// TwinCAT 3 PLC project PLC_851
// Title: 2505
// Company: Infineon
// Author: Utz
// ProgramVersion: 3.1.4023.0
// CompilerDefines: VISU_USEPROPERTYINFO
// libraries:
//   GeneralLib, * (IB-Muhr)
//   CmpBitmapPool, * (System)
//   GeneralLib, * (IB-Muhr)
//   Tc2_EtherCAT, * (Beckhoff Automation GmbH)
//   Tc2_MC2, * (Beckhoff Automation GmbH)
//   Tc2_SerialCom, * (Beckhoff Automation GmbH)
//   Tc2_Standard, * (Beckhoff Automation GmbH)
//   Tc2_System, * (Beckhoff Automation GmbH)
//   Tc2_TcpIp, * (Beckhoff Automation GmbH)
//   Tc2_Utilities, * (Beckhoff Automation GmbH)
//   Tc2_XmlDataSrv, * (Beckhoff Automation GmbH)
//   Tc3_Database, * (Beckhoff Automation GmbH)
//   Tc3_EventLogger, * (Beckhoff Automation GmbH)
//   Tc3_IotBase, * (Beckhoff Automation GmbH)
//   Tc3_Module, * (Beckhoff Automation GmbH)
//   VisuDialogs, * (System)
//   VisuSymbols, * (System)
//   Tc2_Standard,3.3.3.0,Beckhoff Automation GmbH
//   VisuSymbols,3.5.10.0,System
// project tree:
//   DUTs/ ST_RECIPE_ENDURANCE_RUN.TcDUT, ST_RECIPE_BREAK_PRESSURE.TcDUT, ST_RECIPE_GENERAL.TcDUT, ST_RECIPE_LEAK_TEST1.TcDUT, ST_RECIPE_LEAK_TEST2.TcDUT, ST_RECIPE_PARAMS.TcDUT, ST_RECIPE_CYL.TcDUT, ST_SETTINGS.TcDUT
//   FUNCTIONS/FUNCTIONS/MATH/ F_RoundLREAL.TcPOU, F_RoundREAL.TcPOU
//   / GlobalTextList.TcGTLO, GVL.TcGVL, GVL_EventLogger.TcGVL, MeasureTask.TcTTO, PlcTask.TcTTO, ProjectInfo.TcGVL, TXT_LIST_OBJECTS.TcTLO, VisuTask.TcTTO
//   MODULE/ACTOR_VALVE/GENERAL/DUT/ E_POS_STATE.TcDUT, E_SPEED_TYPE.TcDUT, E_PRESSURE_TYPE.TcDUT, ST_CYL_CALIBRATION.TcDUT, ST_HMI_CYLINDER.TcDUT, ST_HMI_VALVE.TcDUT, ST_RECORD.TcDUT, ST_RECORD_DATA.TcDUT
//   MODULE/ACTOR_VALVE/HYDRAULIC_ACTOR/DUT/ E_SEQ_CYLINDER.TcDUT, E_SEQ_ENGINE.TcDUT
//   MODULE/ACTOR_VALVE/HYDRAULIC_ACTOR/ITF/ I_CYLINDER_DA_COUNTER.TcIO, I_CYLINDER_DA_GENERAL.TcIO, I_CYLINDER_DA_TESTDEV2_4.TcIO, I_CYLINDER_SA_GENERAL.TcIO, I_CYLINDER_DA_TESTDEV1.TcIO, I_ENGINE.TcIO, I_PUMP.TcIO, I_PUMP_WITH_BYPASS.TcIO
//   MODULE/ACTOR_VALVE/HYDRAULIC_ACTOR/POU/ FB_CYLINDER_DA_COUNTER.TcPOU, FB_CYLINDER_DA_TESTDEV1.TcPOU, FB_CYLINDER_DA_TESTDEV2_4.TcPOU, FB_PUMP.TcPOU, FB_PUMP_WITH_BYPASS.TcPOU
//   MODULE/ACTOR_VALVE/PNEUMATIC_ACTOR/DUT/ E_PNEU_VAC_VALVE.TcDUT
//   MODULE/ACTOR_VALVE/PNEUMATIC_ACTOR/ITF/ I_PNEU_ACTOR.TcIO, I_STOP_GATE.TcIO, I_VAC_VALVE.TcIO
//   MODULE/ACTOR_VALVE/PNEUMATIC_ACTOR/POU/ FB_STOP_GATE.TcPOU, FB_VAC_BLOW_VALVE.TcPOU, FB_VAC_VALVE.TcPOU, FB_VISU_CYLINDER.TcPOU, FB_VISU_STOP_GATE.TcPOU, FB_VISU_VAC_VALVE.TcPOU, FB_ZYLINDER_TWO_WAY.TcPOU, FB_ZYLINDER_TWO_WAY_MID_POS.TcPOU
//   MODULE/ACTOR_VALVE/PNEUMATIC_ACTOR/TXTLIST/ TXT_LIST_PNEMATIC_ACTOR.TcTLO
//   MODULE/ACTOR_VALVE/PNEUMATIC_ACTOR/VISU/ VisuCylinderGripperDown.TcVIS, VisuCylinderHorLeft.TcVIS, VisuCylinderHorLeftCtrl.TcVIS, VisuCylinderHorRight.TcVIS, VisuCylinderHorRightCtrl.TcVIS, VisuCylinderHorRight_MidPos.TcVIS, VisuCylinderTurn.TcVIS, VisuCylinderVertDown.TcVIS, VisuCylinderVertDownCtrl.TcVIS, VisuCylinderVertUp.TcVIS, VisuCylinderVertUpCtrl.TcVIS
//   MODULE/ACTOR_VALVE/VALVE/DUT/ E_SEQ_VALVE.TcDUT
//   MODULE/ACTOR_VALVE/VALVE/ITF/ I_ENGINE_VALVE.TcIO, I_PRV_PROP.TcIO, I_VALVE_X_3_PROP.TcIO, I_VALVE_X_2.TcIO, I_VALVE_X_3.TcIO
//   MODULE/ACTOR_VALVE/VALVE/POU/ FB_SHUTOFF_VALVE.TcPOU, FB_PRV_PROP.TcPOU, FB_VALVE_X_2.TcPOU, FB_VALVE_X_3.TcPOU, FB_VALVE_X_3_PROP.TcPOU
//   MODULE/BUS_DIAG/POU/ FB_EC_MASTER.TcPOU, FB_VISU_BUS_DIAG.TcPOU
//   MODULE/BUS_DIAG/VISU/ VISU_BUS_DIAG_MASTER.TcVIS
//   MODULE/BYTES_TO_WORD/DUT/ U_BytesToWord.TcDUT
//   MODULE/BYTES_TO_WORD/ITF/ I_WORD_TO_BYTES.TcIO
//   MODULE/BYTES_TO_WORD/POU/ FB_BYTES_TO_WORD.TcPOU, FB_WORD_TO_BYTES.TcPOU
//   MODULE/BYTES_TO_WORD/VISU/ FB_VISU_WORD_TO_BYTES.TcPOU, VISU_WORD_TO_BYTES.TcVIS
//   MODULE/DATABASE/DUT/ E_SEQ_DATABASE.TcDUT, ST_DATABASE_RECORD.TcDUT
//   MODULE/DATABASE/ITF/ I_DATABASE.TcIO, I_INFLUXDB_ADS.TcIO
//   MODULE/DATABASE/POU/ FB_INFLUX_DB.TcPOU, FB_INFLUX_DB_ADS.TcPOU, FB_MY_SQL.TcPOU
//   MODULE/FREQUENCE/ITF/ I_FREQ_GEN.TcIO
//   MODULE/FREQUENCE/POU/ FB_FREQENCE.TcPOU
//   MODULE/GENERAL/DUT/ E_STEP_STATE.TcDUT
//   MODULE/GENERAL/ E_Direction.TcDUT, F_Lineare_Regression.TcPOU, F_RangeSetpoint.TcPOU, stMesswerte.TcDUT, stRampAnalytic.TcDUT, ST_CHART.TcDUT
//   MODULE/GENERAL/INPUTS/ITF/ I_BINARY_SWITCH_SENS.TcIO
//   MODULE/GENERAL/INPUTS/POU/ FB_BINARY_SWITCH_SENS.TcPOU
//   MODULE/GENERAL/SIMU_ANALOG_IN/ FB_SIMU_ANALOG_IN.TcPOU, I_SIMU_ANALOG_IN.TcIO
//   MODULE/HMI/DUT/ E_SEQ_HMI.TcDUT
//   MODULE/HMI/ITF/ I_HMI_CTRL.TcIO
//   MODULE/HMI/POU/ FB_HMI_CTRL.TcPOU, FB_HMI_CTRL_ADS.TcPOU
//   MODULE/SAFETY/DUT/ E_STEP_STATE_ESTOP.TcDUT
//   MODULE/SAFETY/ GVL_SAFETY.TcGVL
//   MODULE/SAFETY/ITF/ I_ESTOP.TcIO
//   MODULE/SAFETY/PIC/ IMG_LIST_GATE_LOCK.TcIPO (not stored)
//   MODULE/SAFETY/POU/ FB_ESTOP.TcPOU
//   MODULE/SAFETY/VISU/ FB_VISU_GATE_LOCK.TcPOU
//   IMPLICIT_CHECKS/ CheckBounds.TcPOU, CheckDivDInt.TcPOU, CheckDivLInt.TcPOU, CheckDivLReal.TcPOU, CheckDivReal.TcPOU, CheckLRangeSigned.TcPOU, CheckLRangeUnsigned.TcPOU, CheckPointer.TcPOU, CheckRangeSigned.TcPOU, CheckRangeUnsigned.TcPOU
//   MODULE/TRAFFIC_LIGHT/ITFs/ I_TrafficLight.TcIO
//   MODULE/TRAFFIC_LIGHT/POUs/ FB_TrafficLight.TcPOU
//   ORGANISATION/DATE_TIME/ITF/ I_CLOCK.TcIO
//   ORGANISATION/DATE_TIME/POU/ FB_CLOCK.TcPOU
//   ORGANISATION/EVENT_LOGGER/ITFs/ I_EVENT_LOGGER.TcIO
//   ORGANISATION/EVENT_LOGGER/POUs/ FB_EVENT_LOGGER.TcPOU
//   ORGANISATION/GENERAL/DUT/ E_SEQ_GENERAL.TcTLEO, E_STEP_STATE_TYPE.TcDUT, ST_GENERAL_HMI.TcDUT, ST_LAST_STEPS.TcDUT, ST_SEQ_CTRL_GEN.TcDUT
//   ORGANISATION/GENERAL/ITF/ FB_Abstract_FunktionCtrl.TcPOU, I_FunctionCtrl.TcIO, I_GENERAL.TcIO
//   ORGANISATION/GENERAL/POU/ FB_GENERAL.TcPOU, F_CreateObjectName.TcPOU
//   ORGANISATION/OP_MODE/DUT/ ST_EVENT_DATA.TcDUT, ST_LOG_EVENT.TcDUT
//   ORGANISATION/OP_MODE/GVL_PARA/ OP_MODE.TcGVL
//   ORGANISATION/OP_MODE/ITF/ I_OP_MODE.TcIO, I_OP_MODE_PAUSE.TcIO, I_OP_MODE_PAUSE_VISU.TcIO
//   ORGANISATION/OP_MODE/POU/ FB_OP_MODE.TcPOU, FB_OP_MODE_HMI.TcPOU, FB_OP_MODE_PAUSE.TcPOU, FB_OP_MODE_PAUSE_VISU.TcPOU, FB_OP_MODE_VISU.TcPOU
//   ORGANISATION/OP_MODE/TXTLIST/ TXT_LIST_OP_MODE.TcTLO
//   ORGANISATION/USER_MANAGER/POU/ FB_ESTOP_RESET.TcPOU
//   POUs/ F_SEND_EVENTLOGGER_MSG.TcPOU, MAIN.TcPOU
//   PROGRAMS/ PrgMeasure.TcPOU, PrgOrg.TcPOU, PrgStation.TcPOU, PrgVisu.TcPOU
//   SUBSTATION/ GVL_SUBSTATION.TcGVL
//   SUBSTATION/STATION_NEST/DUT/ E_SEQ_PROCESS.TcDUT, ST_ENDURANCERUN_RECORD.TcDUT
//   SUBSTATION/STATION_NEST/ GVL_PROCESS.TcGVL
//   SUBSTATION/STATION_NEST/ITF/ I_PROCESS_MAIN.TcIO, I_PROCESS_NEST1.TcIO, I_PROCESS_NEST2_4.TcIO
//   SUBSTATION/STATION_NEST/POU/ FB_PROCESS_MAIN.TcPOU, FB_SEQ_PROCESS_NEST1.TcPOU, FB_SEQ_PROCESS_NEST2_4.TcPOU

CONFIGURATION PLC_851
    RESOURCE PLC ON TwinCAT3
        TASK MeasureTask(INTERVAL := T#10ms, PRIORITY := 2);
        TASK PlcTask(INTERVAL := T#10ms, PRIORITY := 21);
        TASK VisuTask(INTERVAL := T#100000us, PRIORITY := 1);
        PROGRAM PrgMeasure WITH MeasureTask : PrgMeasure;
        PROGRAM PrgStation WITH PlcTask : PrgStation;
        PROGRAM PrgOrg WITH PlcTask : PrgOrg;
        PROGRAM PrgVisu WITH VisuTask : PrgVisu;
    END_RESOURCE
END_CONFIGURATION

// ---- DUTs/ST_RECIPE_ENDURANCE_RUN.TcDUT
TYPE ST_RECIPE_ENDURANCE_RUN :
STRUCT
  // Enables
  bEnableVentCylinder:            BOOL;
  bEnableEnduranceRun:            BOOL;
  bEnableLeakTest1:               BOOL;
  // Vent cylinder
  uiVentCycles:                   UINT;
  // Profiles - Endurance run
  rSpeedA:                        REAL;         // Speed A
  rSpeedB:                        REAL;         // Speed B
  rWorkPressureA:                 REAL;         // Work pressure testing cylinder A
  rWorkPressureB:                 REAL;         // Work pressure testing cylinder B
  rWorkForceA:                    REAL;         // Work force testing cylinder A
  rWorkForceB:                    REAL;         // Work force testing cylinder B
  udiCycles:                      UDINT;        // Count of cycles
  rLoadPressureA:                 REAL;         // Load pressure A (counterload)
  rLoadPressureB:                 REAL;         // Load pressure B (counterload)
  rLoadForceA:                    REAL;         // Load force A (counterload)
  rLoadForceB:                    REAL;         // Load force B (counterload)
  rTurningPointHP:                REAL;         // Cylinder turning point in HP
  rTurningPointWP:                REAL;         // Cylinder turning point in WP
  rDelay:                         REAL;         // Delay on turning point
  // Quick leak test 1 parameter
  udiLT1_Interval:                UDINT;        // Interval for quick leak test 1
  stLT1_Params:                   ST_RECIPE_LEAK_TEST1;
  //rLT1_RestDelay:                 REAL;         // Rest delay aufter test
  //rLT1_LoadForceA:                REAL;         // Load force A (counterload)
  //rLT1_LoadForceB:                REAL;         // Load force B (counterload)
  //rLT1_LoadPressureA:             REAL;         // Testing pressure A for leak test 1
  //rLT1_LoadPressureB:             REAL;         // Testing pressure B for leak test 1
  //uiLT1_DurationPerTest:          UINT;         // Testing duration per test in min
  //rLT1_DistanceBeforeEndPosHP:    REAL;         // Distance to the end position HP
  //rLT1_DistanceBeforeEndPosWP:    REAL;         // Distance to the end position WP
  //rLT1_NokLimit:                  REAL;         // Delta length limit to abort program
END_STRUCT
END_TYPE

// ---- DUTs/ST_RECIPE_BREAK_PRESSURE.TcDUT
TYPE ST_RECIPE_BREAK_PRESSURE :
STRUCT
  // Enables
  bEnableVentCylinder:            BOOL;
  bEnableBreakPressureDet:        BOOL;
  // Vent cylinder
  uiVentCycles:                   UINT;
  // Break pressure determination
  rMinSpeedInMmPerS:              REAL;         // Minimal speed in mm/s
  rEndPosTol:                     REAL;         // End position tolerance
  rIncreaseInterval:              REAL;         // Interval in seconds
  rIncreaseValueInBar:            REAL;         // Value in bar to increase if not mooving
  rNokLimit:                      REAL;         // Pressure limit to abort
END_STRUCT
END_TYPE

// ---- DUTs/ST_RECIPE_GENERAL.TcDUT
TYPE ST_RECIPE_GENERAL :
STRUCT
  uiVentCycles:                   UINT;         // Count of vent cycles
  rVentDelay:                     REAL;         // Delay on HP/WP
  rStrokeLengthDetDelay:          REAL;         // Delay timer to determine stroke length
  rStrokeLengthDetTol:            REAL;         // Stroke length determine tolerance
  rPressureMin:                   REAL;         // Minimum pressure limit
  rPressureMax:                   REAL;         // Maximum pressure limit
  iTemperatureMin:                INT;          // Minimum temperature limit
  iTemperatureMax:                INT;          // Maximum temperature limit
END_STRUCT
END_TYPE

// ---- DUTs/ST_RECIPE_LEAK_TEST1.TcDUT
TYPE ST_RECIPE_LEAK_TEST1 :
STRUCT
  // Enables
  bEnableVentCylinder:            BOOL;
  bEnableLeakTest1:               BOOL;
  // Vent cylinder
  uiVentCycles:                   UINT;
  // Leak test 1
  rRestDelay:                     REAL;         // Rest delay between cycles
  rLoadPressureA:                 REAL;         // Testing pressure A for leak test 1
  rLoadPressureB:                 REAL;         // Testing pressure B for leak test 1
  rLoadForceA:                    REAL;         // Testing force A for leak test 1
  rLoadForceB:                    REAL;         // Testing force B for leak test 1
  udiDurationPerTest:             UDINT;        // Testing duration per test
  rDistanceBeforeEndPosHP:        REAL;         // Distance to the end position HP
  rDistanceBeforeEndPosWP:        REAL;         // Distance to the end position WP
  rNokLimit:                      REAL;         // Delta length limit to abort program
END_STRUCT
END_TYPE

// ---- DUTs/ST_RECIPE_LEAK_TEST2.TcDUT
TYPE ST_RECIPE_LEAK_TEST2 :
STRUCT
  // Enables
  bEnableVentCylinder:            BOOL;
  bEnableLeakTest2:               BOOL;
  // Vent cylinder
  uiVentCycles:                   UINT;
  // Leak test 1
  rRestDelay:                     REAL;         // Rest delay between cycles
  rLoadPressureA:                 REAL;         // Testing pressure A for leak test 2
  rLoadPressureB:                 REAL;         // Testing pressure A for leak test 2
  rLoadForceA:                    REAL;         // Testing force A for leak test 2
  rLoadForceB:                    REAL;         // Testing force A for leak test 2
  udiDurationPerTest:             UDINT;         // Testing duration
  rNokLimit:                      REAL;         // Limit value for abort program
END_STRUCT
END_TYPE

// ---- DUTs/ST_RECIPE_PARAMS.TcDUT
TYPE ST_RECIPE_PARAMS :
STRUCT
  /// Cylinder parameter
  stRecipeCyl:            ST_RECIPE_CYL;
  /// Profiles - Endurance run
  stRecipeEnduranceRun:   ST_RECIPE_ENDURANCE_RUN;
  /// Profiles - General settings
  stRecipeGeneral:        ST_RECIPE_GENERAL;
  /// Profiles - Leak test 1
  stRecipeLeakTest1:      ST_RECIPE_LEAK_TEST1;
  /// Profiles - Leak test 2
  stRecipeLeakTest2:      ST_RECIPE_LEAK_TEST2;
  /// Profiles - Determine break pressure
  stRecipeBreakPressure:  ST_RECIPE_BREAK_PRESSURE;
END_STRUCT
END_TYPE

// ---- DUTs/ST_RECIPE_CYL.TcDUT
TYPE ST_RECIPE_CYL :
STRUCT
  sItemName:              STRING;       // Name of the cylinder
  sItemNumber:            STRING;       // Item number of the cylinder
  bDoubleActing:          BOOL;         // Double- or singleacting cylinder
  rStrokeLength:          REAL;         // The theoretical Stroke length
  rStrokeLengthTol:       REAL;         // Stroke length tolerance
  lrPistonSurfaceA:       LREAL;        // Piston surface for the working direction
  lrPistonSurfaceB:       LREAL;        // Piston surface for the homing direction
  rMaxPremittedPressure:  REAL;         // Maximum allowable pressure
  sInfo:                  STRING;       // Other
END_STRUCT
END_TYPE

// ---- DUTs/ST_SETTINGS.TcDUT
TYPE ST_SETTINGS :
STRUCT
  // Control outside the HMI
  bCloseHmi:                      BOOL;
  bShutdownPc:                    BOOL;
  bRestartPc:                     BOOL;
  bShowWinKeyboard:               BOOL;
  // Speed regulation and max speed efficiency
  rSpeedEfficiencyFactor:         REAL;
  rSpeedRegulationFactor:         REAL;
  rSpeedRegulationTolerance:      REAL;
  // Pressure regulation
  rPressureRegulationFactor:      REAL;
  rPressureRegulationTolerance:   REAL;
  
  // Recording
  uiRecordDelay:                  UINT;
END_STRUCT
END_TYPE

// ---- MODULE/ACTOR_VALVE/GENERAL/DUT/E_POS_STATE.TcDUT
{attribute 'qualified_only'}
{attribute 'strict'}
TYPE E_POS_STATE :
(
	InBasePos,
	InWorkPos,
	InMidPos,
	InBasePosValveOff,
	InWorkPosValveOff,
	NoDefPos,
	MoveToBase,
	MoveToWork,
	TimeOutToWork,
	TimeOutToBase,
	MoveToBaseLock,
	MoveToWorkLock
);
END_TYPE

// ---- MODULE/ACTOR_VALVE/GENERAL/DUT/E_SPEED_TYPE.TcDUT
{attribute 'qualified_only'}
{attribute 'strict'}
TYPE E_SPEED_TYPE :
(
	MM_PER_SECOND,
  PERCENT
);
END_TYPE

// ---- MODULE/ACTOR_VALVE/GENERAL/DUT/E_PRESSURE_TYPE.TcDUT
{attribute 'qualified_only'}
{attribute 'strict'}
TYPE E_PRESSURE_TYPE :
(
  VALUE,
	BAR,
  FORCE,
  PERCENT
);
END_TYPE

// ---- MODULE/ACTOR_VALVE/GENERAL/DUT/ST_CYL_CALIBRATION.TcDUT
TYPE ST_CYL_CALIBRATION :
STRUCT
  uiValue:          UINT;
  uiPressure:       UINT;
  uiState:          UINT;
END_STRUCT
END_TYPE

// ---- MODULE/ACTOR_VALVE/GENERAL/DUT/ST_HMI_CYLINDER.TcDUT
TYPE ST_HMI_CYLINDER :
STRUCT    
  // OP mode
  itfOpMode:			        I_OP_MODE;
                 
  // Control              
  bToHPTriggered:         BOOL;
  bToWPTriggered:         BOOL;
  bToSetPosTriggered:     BOOL;
  bStopTriggered:         BOOL;
  uiSpeedInPercent:       UINT;
  lrPosToSet:             LREAL;
  
  // Info
  lrMinPosVal:            LREAL;
  lrMaxPosVal:            LREAL;
  lrCurrentPos:           LREAL;
  bInWP:                  BOOL;
  bInHP:                  BOOL;
  sState:                 STRING;
  bPressureOk:            BOOL;
  rPressure:              REAL;
END_STRUCT
END_TYPE

// ---- MODULE/ACTOR_VALVE/GENERAL/DUT/ST_HMI_VALVE.TcDUT
TYPE ST_HMI_VALVE :
STRUCT
  // OP mode
  itfOpMode:			        I_OP_MODE;
                 
  // Control              
  bToHP:                  BOOL;
  bToWP:                  BOOL;
  bToSetPos:              BOOL;
  uiSpeedInPercent:       UINT;
  lrPosToSet:             LREAL;
  
  // Info
  sState:                 STRING;
  bPressureOk:            BOOL;
  diPressure:             DINT;
END_STRUCT
END_TYPE

// ---- MODULE/ACTOR_VALVE/GENERAL/DUT/ST_RECORD.TcDUT
TYPE ST_RECORD :
STRUCT
	listRecordData:		ARRAY[0..2999] OF ST_RECORD_DATA;
END_STRUCT
END_TYPE

// ---- MODULE/ACTOR_VALVE/GENERAL/DUT/ST_RECORD_DATA.TcDUT
TYPE ST_RECORD_DATA:
STRUCT
	rPosition:		    REAL;
	rPressureInBar:		REAL;
END_STRUCT
END_TYPE

// ---- MODULE/ACTOR_VALVE/HYDRAULIC_ACTOR/DUT/E_SEQ_CYLINDER.TcDUT
{attribute 'qualified_only'}
{attribute 'strict'}
TYPE E_SEQ_CYLINDER :
(
	// GENERAL STEPS
	BASE := 0,
  INIT,
  SETUP,
  // Process
  SET_MAX_POS,
  SET_SPEED_BWD,
  SET_SPEED_FWD,
  SET_WORK_PRESSURE,
  SET_WORK_PRESSURE_ZERO,
  SET_ZERO_POS,
  STOP,
  STOP_AND_LOCK,
  TO_HP,
  TO_SET_POS,
  TO_WP,
  PRESSURE_CALIBRATION,
  LOW_PRESSURE_CALIBRATION,
  LOW_PRESSURE_CIRCUIT,
  LOW_PRESSURE_MODE,
  OPEN_RESERVOIR,
  OPEN_LOCK_VALVES,
  PUMP2_ADD,
  PUMP3_ADD,
  PUMP4_ADD,
  
  END,
	ERROR_SEQ	
);
END_TYPE

// ---- MODULE/ACTOR_VALVE/HYDRAULIC_ACTOR/DUT/E_SEQ_ENGINE.TcDUT
{attribute 'qualified_only'}
{attribute 'strict'}
TYPE E_SEQ_ENGINE :
(
	// GENERAL STEPS
	BASE := 0,
  INIT,
  SETUP,
  // Process
  ON,
  OFF,
  OPEN,
  CLOSE,
  BYPASS,
  
  END,
	ERROR_SEQ	
);
END_TYPE

// ---- MODULE/ACTOR_VALVE/PNEUMATIC_ACTOR/DUT/E_PNEU_VAC_VALVE.TcDUT
{attribute 'qualified_only'}
{attribute 'strict'}
TYPE E_PNEU_VAC_VALVE :
(
	VacDetect,
	Vac_ON_NotDetect,
	AllOff,
	Blowing
);
END_TYPE

// ---- MODULE/ACTOR_VALVE/VALVE/DUT/E_SEQ_VALVE.TcDUT
{attribute 'qualified_only'}
{attribute 'strict'}
TYPE E_SEQ_VALVE :
(
	// GENERAL STEPS
	BASE := 0,
  INIT,
  WAIT_FOR_AUTOMATIC_START,
  SETUP,
  
  // Process
	SET_HP,
	SET_WP1,
  SET_WP2,
  SET_LIMIT,
  SET_LIMIT_SMOOTH,
  
  END,
	ERROR_SEQ	
);
END_TYPE

// ---- MODULE/BYTES_TO_WORD/DUT/U_BytesToWord.TcDUT
TYPE U_BytesToWord :
UNION
	arByteIn:ARRAY [0..1] OF BYTE;
	uintOut: UINT;
END_UNION
END_TYPE

// ---- MODULE/DATABASE/DUT/E_SEQ_DATABASE.TcDUT
{attribute 'qualified_only'}
{attribute 'strict'}
{attribute 'to_string'}
TYPE E_SEQ_DATABASE :
(
	// GENERAL STEPS
	BASE := 0,
  INIT,
  WAIT_FOR_AUTOMATIC_START,
  SETUP,
  // Process
  CREATE_DATABASE,
	CONNECT,
  EXECUTE_SIMPLIFY_CMD,
  EXECUTE_CMD,
  CREATE_TABLE,
  WRITE,
  WRITE_STRUCT,
  WRITE_BY_SYMBOL,
  OVERWRITE,
  READ,
  READ_STRUCT,
  CLEAR_TABLE,
  DELETE_TABLE,
  DISCONNECT,
  TABLE_EXIST_CHECK,
  
  // InfluxDB per ADS
  BUCKET_EXIST_CHECK,
  MEASUREMENT_EXIST_CHECK,
  TAG_EXIST_CHECK,
  FIELD_EXIST_CHECK,
  CLEAR_MEASUREMENT,
  DELETE_ALL_MEASUREMENTS,
  DELETE_MEASUREMENT,
  DELETE_TAG,
  DELETE_TAG_CONTENT_BLOCK,
  DELETE_FIELD,
  GET_TOTAL_MEASUREMENTS,
  
  END,
	ERROR_SEQ	
);
END_TYPE

// ---- MODULE/DATABASE/DUT/ST_DATABASE_RECORD.TcDUT
TYPE ST_DATABASE_RECORD :
STRUCT
  sTimeStamp:                         T_MaxString;
  sTimer:                             T_MaxString;
  liTargetCycles:                     LINT;
  liActiveCycle:                      LINT;
  iTestDirection:                     SINT;
  rTargetTestPressureInBarA:          REAL;
  rTargetTestPressureInBarB:          REAL;
  rCurrentTestPressureInBar:          REAL;
  rTargetTestForceInKNA:              REAL;
  rTargetTestForceInKNB:              REAL;
  rCurrentTestForceInKN:              REAL;
  rTestPressureAInBar:                REAL;
  rTestPressureBInBar:                REAL;
  rBreakawayPressureInBar:            REAL;
  rBreakawayPressureAInBar:           REAL;
  rBreakawayPressureBInBar:           REAL;
  rReservoirPressureInBar:            REAL;
  rTargetCounterPressureInBarA:       REAL;
  rTargetCounterPressureInBarB:       REAL;
  rCurrentCounterPressureInBar:       REAL;
  rTargetCounterForceInKNA:           REAL;
  rTargetCounterForceInKNB:           REAL;
  rCurrentCounterForceInKN:           REAL;
  lrPosition:                         LREAL;
  lrPositionMin:                      LREAL;
  lrPositionMax:                      LREAL;
  lrCylStrokeLength:                  LREAL;
  lrTemperature:                      LREAL;
  lrCylPistonSurfaceA:                LREAL;
  lrCylPistonSurfaceB:                LREAL;
  lrNokLimit:                         LREAL;
  lrCurrentNokDifference:             LREAL;
  lrCurrentNokLimitInPercent:         LREAL;
  lrTargetSpeedAInMmPerS:             LREAL;
  lrTargetSpeedBInMmPerS:             LREAL;
  lrCurrentSpeedInMmPerS:             LREAL;
END_STRUCT
END_TYPE

// ---- MODULE/GENERAL/DUT/E_STEP_STATE.TcDUT
{attribute 'qualified_only'}
{attribute 'strict'}
TYPE E_STEP_STATE :
(
	//GENERAL STEPS
	BASE := 0,
  INIT,
  RESET,
  
  SET_READY,
	SET_BUSY,
  SET_DONE,
  
  ERROR := 999
);
END_TYPE

// ---- MODULE/GENERAL/E_Direction.TcDUT
{attribute 'qualified_only'}
{attribute 'strict'}
TYPE E_Direction :
(
	Forward:=0,
	Backward,
	Clockwise,
	Counterclockwise
);
END_TYPE

// ---- MODULE/GENERAL/stMesswerte.TcDUT
TYPE stMesswerte :
STRUCT
	X: 			LREAL;
	Y: 			LREAL;
	//SQR_Y_Ys:	LREAL;
	//sqr_Y_Yd:  	LREAL;
END_STRUCT
END_TYPE

// ---- MODULE/GENERAL/stRampAnalytic.TcDUT
TYPE stRampAnalytic :
STRUCT
	lrExp2R: 	LREAL;
	lrGain:		LREAL;
	lrOffset:	LREAL;
END_STRUCT
END_TYPE

// ---- MODULE/GENERAL/ST_CHART.TcDUT
TYPE ST_CHART :
STRUCT
  sName0:        STRING;
  diValue0:      DINT;
  sName1:        STRING;
  diValue1:      DINT;
  sName2:        STRING;
  diValue2:      DINT;
  sName3:        STRING;
  diValue3:      DINT;
  sName4:        STRING;
  diValue4:      DINT;
  sName5:        STRING;
  diValue5:      DINT;
  sName6:        STRING;
  diValue6:      DINT;
  sName7:        STRING;
  diValue7:      DINT;
  sName8:        STRING;
  diValue8:      DINT;
  sName9:        STRING;
  diValue9:      DINT;
END_STRUCT
END_TYPE

// ---- MODULE/HMI/DUT/E_SEQ_HMI.TcDUT
{attribute 'qualified_only'}
{attribute 'strict'}
{attribute 'to_string'}
TYPE E_SEQ_HMI :
(
	// GENERAL STEPS
	BASE := 0,
  INIT,
  WAIT_FOR_AUTOMATIC_START,
  SETUP,
  // Process
  START_HMI,
  CLOSE_HMI,
  PC_REBOOT,
  PC_SHUTDOWN,
  SHOW_WIN_KEYBOARD,
  HIDE_WIN_KEYBOARD,
  
  END,
	ERROR_SEQ	
);
END_TYPE

// ---- MODULE/SAFETY/DUT/E_STEP_STATE_ESTOP.TcDUT
{attribute 'qualified_only'}
{attribute 'strict'}
TYPE E_STEP_STATE_ESTOP :
(
	//GENERAL STEPS
	BASE := 0,
	RESET,
	START_INIT,
	
	INIT_BUSY,
	INIT_TURN_OFF_CYLINDER,
	INIT_DONE,
	START_SEQ,
	DEBUG_BREAK,
	
	ESTOP_OK,
	ESTOP_PRESSED,
	WAIT_QUIT_ESTOP,
	SET_QUIT_ESTOP,
	RESET_QUIT_ESTOP,
	ESTOP_QUIT_OK,
	
	TIME_OUT,
	TIME_OUT_TO_QUIT,
	ERROR,
	ERROR_TO_QUIT,
	ERROR_RESTART,
	IBN_DUMMY,
	//SPECIFIC STEPS
	START_LAST_TEST
);
END_TYPE

// ---- ORGANISATION/GENERAL/DUT/E_SEQ_GENERAL.TcTLEO
{attribute 'qualified_only'}
{attribute 'strict'}
{attribute 'to_string'}
TYPE E_SEQ_GENERAL :
(
	READY,
	EXECUTE,
	RESET,
	BUSY,
	DONE,
	ERROR,
	TIME_OUT	
);
END_TYPE

// ---- ORGANISATION/GENERAL/DUT/E_STEP_STATE_TYPE.TcDUT
{attribute 'qualified_only'}
{attribute 'strict'}
TYPE E_STEP_STATE_TYPE :
(
	BASE := 0,
	RESET,
	INIT,
	INIT_OK,
	INIT_RUN,			
	WAIT_RUN,			
	WAIT_USER_ACTION, 	
	RUN,					
	ERROR_RUN,			
	ERROR,				
	RUN_ALWAYS		
	            	
);
END_TYPE

// ---- ORGANISATION/GENERAL/DUT/ST_GENERAL_HMI.TcDUT
TYPE ST_GENERAL_HMI :
STRUCT
	strObjectName:  STRING;
	strActiveState: STRING;
	xErrorState:    WORD;
	bEnableCtrl:    BOOL;
	
END_STRUCT
END_TYPE

// ---- ORGANISATION/GENERAL/DUT/ST_LAST_STEPS.TcDUT
TYPE ST_LAST_STEPS :
STRUCT
	strStepName: 		    STRING;
	iStepID:			      INT;
	tStepTime: 			    TIME;
	tDelayTime:			    TIME;
	eStepType:			    BOOL;
	bBreakpointActive: 	BOOL;
	bDisableBreakpoint: BOOL;
END_STRUCT
END_TYPE

// ---- ORGANISATION/GENERAL/DUT/ST_SEQ_CTRL_GEN.TcDUT
TYPE ST_SEQ_CTRL_GEN :
STRUCT
	strObject:												                      STRING;
	strObjectPath:											                    STRING;
	eActiveSeqState:                   						          E_SEQ_GENERAL;
	eLastActiveSeqState:                   					        E_SEQ_GENERAL;
	iInternalSeqStateCase, iLastInternalSeqStateCase:       INT:=-1;       
	tonDelay, tonTimeOut, tonStepTime:						          TON;
	tDelay:													                        TIME := T#100MS;
	tTimeOut:												                        TIME := T#100MS;
	tTimeOutExt:											                      TIME := T#100MS;
	bDelayActive, bTimeOutActiveQuit, bTimeOutActiveNoQuit:	BOOL;//Timer Option
	bActiveStep, bDebugAcitve, bDebugNext:					        BOOL;//Debug Option
 	iError:													                        INT; //ERROR-CODE                    	                   		
	listLastSteps:											                    ARRAY[0..49] OF ST_LAST_STEPS;	
	strExtraInfo:											                      STRING; 
	eStep_Type:												                      E_STEP_STATE_TYPE; 
	bDebugModeActive:										                    BOOL;   
	bWaitForBreakpoint:										                  BOOL;
	bBreakpointActive:										                  BOOL;
	bDebugResume:											                      BOOL;   
	listBreakpoint:											                    ARRAY[0..10] OF  INT;  
  bExitSetReadyState:                                     BOOL;
END_STRUCT
END_TYPE

// ---- ORGANISATION/OP_MODE/DUT/ST_EVENT_DATA.TcDUT
TYPE ST_EVENT_DATA :
STRUCT
		String1: STRING;
		String2: STRING;
END_STRUCT
END_TYPE

// ---- ORGANISATION/OP_MODE/DUT/ST_LOG_EVENT.TcDUT
TYPE ST_LOG_EVENT :
STRUCT
	CfgEvent		: TcEvent;
	fbEvent			: ADSLOGEVENT;
	bActive			: BOOL;
	stEventData		: ST_EVENT_DATA;
	strId			: STRING;
	strText			: STRING;
	enuEventType	: ENUM_EVENT_TYPE;
END_STRUCT
END_TYPE

// ---- SUBSTATION/STATION_NEST/DUT/E_SEQ_PROCESS.TcDUT
{attribute 'qualified_only'}
{attribute 'strict'}
{attribute 'to_string'}
TYPE E_SEQ_PROCESS :
(
	//GENERAL STEPS
	BASE := 0,
  AUTOMATIC,
  MANUAL,
  INIT,
  SETUP,
  // Process
	MEASURE_STROKE_LENGTH,
  VENT_CYLINDER,
  MOVE_TO_SET_POS,
  BREAK_PRESSURE_DET,
  LEAK_TEST_1,
  LEAK_TEST_2,
  MAX_SPEED_RECORD,
  ENDURANCE_RUN,
  STOP_ENGINE,
  STOP,
  ESTOP,
  RESET_DISTANCE,
  MOVE_CYL_TO_HP,
  
  END,
	ERROR_SEQ	
);
END_TYPE

// ---- SUBSTATION/STATION_NEST/DUT/ST_ENDURANCERUN_RECORD.TcDUT
TYPE ST_ENDURANCERUN_RECORD :
STRUCT
	id: DINT;
	dtTimeStamp: DT;
	sItem: STRING(255);
	diCycle: DINT;
	rWorkPressure: REAL;
	rLoadPressure: REAL;
	rPosition: REAL;
	rTemperature: REAL;
END_STRUCT
END_TYPE

// ---- GVL.TcGVL
{attribute 'qualified_only'}
VAR_GLOBAL
  
END_VAR

// ---- GVL_EventLogger.TcGVL
{attribute 'qualified_only'}
VAR_GLOBAL
	fbPrevMsg:									TcEventEntry;
	udiPrevMsgId:								UDINT;
END_VAR

// ---- MODULE/SAFETY/GVL_SAFETY.TcGVL
{attribute 'qualified_only'}
VAR_GLOBAL
	bInvisibleLockOpened:										BOOL;
	bInvisibleLockClosed:										BOOL;
	bInvisibleLockClosedAndQuit:								BOOL;
END_VAR

// ---- ORGANISATION/OP_MODE/GVL_PARA/OP_MODE.TcGVL
{attribute 'qualified_only'}
VAR_GLOBAL CONSTANT
	//OP MODE STATE ACTIVE
	AUTO			: INT := 1;
	MANUAL			: INT := 2;
	DEBUG			: INT := 3;
	INIT			: INT := 4;
	INIT_OK			: INT := 5;
	PAUSE			: INT := 6;
  STOP      : INT := 15;
	//OP MODE SECUNDARY
	SAFETY_STOP		: INT := 7;
	MACHINE_ERROR 	: INT := 8;	
	CONTROL_ON		: INT := 9;
	MAIN_AIR_OK		: INT := 10;
	
	//OP MODE STATE TEMPORARY
	AUTO_TEMPORARY	: INT := 11;
	MANUAL_TEMPORARY: INT := 12;
	DEBUG_TEMPORARY	: INT := 13;
	RESET_TEMPORARY	: INT := 14;

END_VAR

// ---- ProjectInfo.TcGVL
{attribute 'qualified_only'}
VAR_GLOBAL CONSTANT
	strProjectNumber: STRING:='3531';
	strProjectMng: STRING:='Stefan Utz';
	strPhone: STRING:='???';
	
END_VAR

// ---- SUBSTATION/GVL_SUBSTATION.TcGVL
{attribute 'qualified_only'}
VAR_GLOBAL
END_VAR

// ---- SUBSTATION/STATION_NEST/GVL_PROCESS.TcGVL
{attribute 'qualified_only'}
VAR_GLOBAL
	
END_VAR

// ---- MODULE/ACTOR_VALVE/HYDRAULIC_ACTOR/ITF/I_CYLINDER_DA_COUNTER.TcIO
INTERFACE I_CYLINDER_DA_COUNTER EXTENDS I_CYLINDER_DA_GENERAL

METHOD M_AutoMode : BOOL
VAR_INPUT
  bEnable:        BOOL;
END_VAR
END_METHOD

METHOD M_LowPressureCircuit : BOOL
VAR_INPUT
  bAdd:               BOOL;
END_VAR
END_METHOD

END_INTERFACE

// ---- MODULE/ACTOR_VALVE/HYDRAULIC_ACTOR/ITF/I_CYLINDER_DA_GENERAL.TcIO
INTERFACE I_CYLINDER_DA_GENERAL EXTENDS I_CYLINDER_SA_GENERAL

METHOD M_ToHP : BOOL
VAR_INPUT
  /// Bar | Force in N | Percent 0-100 | Value 0-32767
  ePressureType:            E_PRESSURE_TYPE;
  rWorkPressure:            REAL;
  bPressureRegulation:      BOOL;
  /// Just need for prop valve
  eSpeedType:               E_SPEED_TYPE;
  rSpeed:                   REAL;
END_VAR
END_METHOD

PROPERTY P_PistonSurfaceB : LREAL
GET
END_GET
END_PROPERTY

END_INTERFACE

// ---- MODULE/ACTOR_VALVE/HYDRAULIC_ACTOR/ITF/I_CYLINDER_DA_TESTDEV2_4.TcIO
INTERFACE I_CYLINDER_DA_TESTDEV2_4 EXTENDS I_CYLINDER_DA_GENERAL

METHOD M_OpenLockValves : BOOL
VAR_INPUT
  bOpenChA:        BOOL;
  bOpenChB:        BOOL;
END_VAR
END_METHOD

METHOD M_SetMaxPos : BOOL
VAR_INPUT
END_VAR
END_METHOD

METHOD M_SetZeroPos : BOOL
VAR_INPUT
END_VAR
END_METHOD

METHOD M_StopAndLock : BOOL
VAR_INPUT
END_VAR
END_METHOD

METHOD M_ToSetPos : BOOL
VAR_INPUT
  lrToSetPos:                 LREAL;
  /// Just need for prop valve
  eSpeedType:               E_SPEED_TYPE;
  rSpeed:                   REAL; 
END_VAR
END_METHOD

PROPERTY P_ActiveDirection : SINT
GET
END_GET
END_PROPERTY

PROPERTY P_DoubleActing : BOOL
GET
END_GET
END_PROPERTY

PROPERTY P_MaxPosVal : LREAL
GET
END_GET
END_PROPERTY

PROPERTY P_MinPosVal : LREAL
GET
END_GET
END_PROPERTY

PROPERTY P_Position : LREAL
GET
END_GET
END_PROPERTY

PROPERTY P_PositionAbs : LREAL
GET
END_GET
END_PROPERTY

PROPERTY P_PressureChA : REAL
GET
END_GET
END_PROPERTY

PROPERTY P_PressureChB : REAL
GET
END_GET
END_PROPERTY

PROPERTY P_SpeedInMmPerSecond : REAL
GET
END_GET
END_PROPERTY

PROPERTY P_SpeedInPercent : LREAL
GET
END_GET
END_PROPERTY

PROPERTY P_StrokeLength : REAL
GET
END_GET
END_PROPERTY

PROPERTY P_StrokeLengthInitialized : BOOL
GET
END_GET
SET
END_SET
END_PROPERTY

END_INTERFACE

// ---- MODULE/ACTOR_VALVE/HYDRAULIC_ACTOR/ITF/I_CYLINDER_SA_GENERAL.TcIO
INTERFACE I_CYLINDER_SA_GENERAL EXTENDS I_GENERAL_OBJECT

METHOD M_PressureCalibration : BOOL
VAR_INPUT
END_VAR
END_METHOD

METHOD M_Reset : BOOL
VAR_INPUT
END_VAR
END_METHOD

METHOD M_SetReady : BOOL
VAR_INPUT
END_VAR
END_METHOD

METHOD M_SetWorkPressure : BOOL
VAR_INPUT
  ePressureType:                   E_PRESSURE_TYPE;
  rWorkPressure:                   REAL;
END_VAR
END_METHOD

METHOD M_SetWorkPressureZero : BOOL
VAR_INPUT
END_VAR
END_METHOD

METHOD M_Stop : BOOL
VAR_INPUT
END_VAR
END_METHOD

METHOD M_ToWP : BOOL
VAR_INPUT
  /// Bar | Force in N | Percent 0-100 | Value 0-32767
  ePressureType:            E_PRESSURE_TYPE;
  rWorkPressure:            REAL;
  bPressureRegulation:      BOOL;
  /// Just need for prop valve
  eSpeedType:               E_SPEED_TYPE;
  rSpeed:                   REAL;
END_VAR
END_METHOD

PROPERTY P_CurrentForceInKN : REAL
GET
END_GET
END_PROPERTY

PROPERTY P_PistonSurfaceA : LREAL
GET
END_GET
END_PROPERTY

PROPERTY P_PressureOk : BOOL
GET
END_GET
END_PROPERTY

PROPERTY P_ReadyState : BOOL
GET
END_GET
END_PROPERTY

PROPERTY P_WorkPressure : REAL
GET
END_GET
END_PROPERTY

END_INTERFACE

// ---- MODULE/ACTOR_VALVE/HYDRAULIC_ACTOR/ITF/I_CYLINDER_DA_TESTDEV1.TcIO
INTERFACE I_CYLINDER_DA_TESTDEV1 EXTENDS I_CYLINDER_DA_TESTDEV2_4

METHOD M_LowPressureCalibration : BOOL
END_METHOD

METHOD M_LowPressureMode : BOOL
VAR_INPUT
  bSet:                            BOOL;
	ePressureType:                   E_PRESSURE_TYPE;
  rWorkPressure:                   REAL;
END_VAR
END_METHOD

METHOD M_OpenReservoir : BOOL
VAR_INPUT
  bOpenA:       BOOL;
  bOpenB:       BOOL;
END_VAR
END_METHOD

METHOD M_Pump2Add : BOOL
VAR_INPUT
  bAdd:         BOOL;
END_VAR
END_METHOD

METHOD M_Pump3Add : BOOL
VAR_INPUT
  bAdd:         BOOL;
END_VAR
END_METHOD

METHOD M_Pump4Add : BOOL
VAR_INPUT
  bAdd:         BOOL;
END_VAR
END_METHOD

PROPERTY P_ActiveVolumeFlow : REAL
GET
END_GET
END_PROPERTY

{warning 'Eigenschaftenimplementierung hinzufügen'}
PROPERTY P_CurrentLowPressureForceInN : REAL
GET
END_GET
END_PROPERTY

PROPERTY P_LowPressure : REAL
GET
END_GET
END_PROPERTY

PROPERTY P_LowPressureChA : REAL
GET
END_GET
END_PROPERTY

PROPERTY P_LowPressureChB : REAL
GET
END_GET
END_PROPERTY

PROPERTY P_LowPressureModeEnable : BOOL
GET
END_GET
END_PROPERTY

PROPERTY P_Pump2Added : BOOL
GET
END_GET
END_PROPERTY

PROPERTY P_Pump3Added : BOOL
GET
END_GET
END_PROPERTY

PROPERTY P_Pump4Added : BOOL
GET
END_GET
END_PROPERTY

PROPERTY P_ReservoirAOpened : BOOL
GET
END_GET
END_PROPERTY

PROPERTY P_ReservoirBOpened : BOOL
GET
END_GET
END_PROPERTY

PROPERTY P_ReservoirPressure : REAL
GET
END_GET
END_PROPERTY

END_INTERFACE

// ---- MODULE/ACTOR_VALVE/HYDRAULIC_ACTOR/ITF/I_ENGINE.TcIO
INTERFACE I_ENGINE EXTENDS I_GENERAL_OBJECT

METHOD M_Off : BOOL
VAR_INPUT
END_VAR
END_METHOD

METHOD M_On : BOOL
VAR_INPUT
END_VAR
END_METHOD

METHOD M_SetReady : BOOL
VAR_INPUT
END_VAR
END_METHOD

PROPERTY P_Busy : BOOL
GET
END_GET
END_PROPERTY

PROPERTY P_ReadyState : BOOL
GET
END_GET
END_PROPERTY

PROPERTY P_State : BOOL
GET
END_GET
END_PROPERTY

END_INTERFACE

// ---- MODULE/ACTOR_VALVE/HYDRAULIC_ACTOR/ITF/I_PUMP.TcIO
INTERFACE I_PUMP EXTENDS I_ENGINE

END_INTERFACE

// ---- MODULE/ACTOR_VALVE/HYDRAULIC_ACTOR/ITF/I_PUMP_WITH_BYPASS.TcIO
INTERFACE I_PUMP_WITH_BYPASS EXTENDS I_ENGINE

METHOD M_Bypass : BOOL
VAR_INPUT
  bEnable:        BOOL;
END_VAR
END_METHOD

PROPERTY P_BypassState : BOOL
GET
END_GET
END_PROPERTY

END_INTERFACE

// ---- MODULE/ACTOR_VALVE/PNEUMATIC_ACTOR/ITF/I_PNEU_ACTOR.TcIO
INTERFACE I_PNEU_ACTOR EXTENDS I_GENERAL_OBJECT

METHOD M_LockMovment
VAR_INPUT
	bLockBaseMovement: 	BOOL;
	bLockWorkMovement: 	BOOL;
	itfObject:			I_GENERAL_OBJECT;
END_VAR
END_METHOD

METHOD M_Stop
VAR_INPUT
END_VAR
END_METHOD

METHOD M_ToBasePos
VAR_INPUT
END_VAR
END_METHOD

METHOD M_ToWorkPos
VAR_INPUT
END_VAR
END_METHOD

METHOD M_UnLockMovment
VAR_INPUT
END_VAR
END_METHOD

PROPERTY P_State : E_POS_STATE
GET
END_GET
END_PROPERTY

PROPERTY P_TimeOutToBase : TIME
GET
END_GET
SET
END_SET
END_PROPERTY

PROPERTY P_TimeOutToWork : TIME
GET
END_GET
SET
END_SET
END_PROPERTY

END_INTERFACE

// ---- MODULE/ACTOR_VALVE/PNEUMATIC_ACTOR/ITF/I_STOP_GATE.TcIO
INTERFACE I_STOP_GATE EXTENDS I_GENERAL_OBJECT

METHOD M_Close
VAR_INPUT
END_VAR
END_METHOD

METHOD M_Open
VAR_INPUT
END_VAR
END_METHOD

METHOD M_Seperate
VAR_INPUT
	iCntCarrier: INT;
END_VAR
END_METHOD

PROPERTY P_CarrierByStopGate : BOOL
GET
END_GET
END_PROPERTY

PROPERTY P_Congestion : BOOL
GET
END_GET
END_PROPERTY

END_INTERFACE

// ---- MODULE/ACTOR_VALVE/PNEUMATIC_ACTOR/ITF/I_VAC_VALVE.TcIO
INTERFACE I_VAC_VALVE EXTENDS I_GENERAL_OBJECT

METHOD M_AllOff
VAR_INPUT
END_VAR
END_METHOD

METHOD M_Blow
VAR_INPUT
END_VAR
END_METHOD

METHOD M_Vac
VAR_INPUT
END_VAR
END_METHOD

PROPERTY P_STATE : E_PNEU_VAC_VALVE
GET
END_GET
END_PROPERTY

END_INTERFACE

// ---- MODULE/ACTOR_VALVE/VALVE/ITF/I_ENGINE_VALVE.TcIO
INTERFACE I_ENGINE_VALVE EXTENDS I_GENERAL_OBJECT

METHOD M_Close : BOOL
VAR_INPUT
END_VAR
END_METHOD

METHOD M_Open : BOOL
VAR_INPUT
END_VAR
END_METHOD

METHOD M_SetReady : BOOL
VAR_INPUT
END_VAR
END_METHOD

PROPERTY P_Closed : BOOL
GET
END_GET
END_PROPERTY

PROPERTY P_Open : BOOL
GET
END_GET
END_PROPERTY

PROPERTY P_ReadyState : BOOL
GET
END_GET
END_PROPERTY

PROPERTY P_Undefined : BOOL
GET
END_GET
END_PROPERTY

END_INTERFACE

// ---- MODULE/ACTOR_VALVE/VALVE/ITF/I_PRV_PROP.TcIO
INTERFACE I_PRV_PROP EXTENDS I_GENERAL_OBJECT

METHOD M_SetLimit : BOOL
VAR_INPUT
  ePressureType:      E_PRESSURE_TYPE;
  rLimit:             REAL;
END_VAR
END_METHOD

METHOD M_SetReady : BOOL
VAR_INPUT
END_VAR
END_METHOD

PROPERTY P_LimitInBar : REAL
GET
END_GET
END_PROPERTY

PROPERTY P_LimitInPercent : REAL
GET
END_GET
END_PROPERTY

PROPERTY P_MaxLimitInBar : REAL
GET
END_GET
END_PROPERTY

PROPERTY P_ReadyState : BOOL
GET
END_GET
END_PROPERTY

END_INTERFACE

// ---- MODULE/ACTOR_VALVE/VALVE/ITF/I_VALVE_X_3_PROP.TcIO
INTERFACE I_VALVE_X_3_PROP EXTENDS I_GENERAL_OBJECT

METHOD M_Reset : BOOL
VAR_INPUT
END_VAR
END_METHOD

METHOD M_SetReady : BOOL
VAR_INPUT
END_VAR
END_METHOD

METHOD M_ValveCtrl : BOOL
VAR_INPUT
  /// -100 to -1 = Move to HP, 1 to 100 = Move to WP, 0 = Off
  rSpeedInPercent:        REAL;
  tDelay:                 TIME;
END_VAR
END_METHOD

METHOD M_ValveCtrlSmooth : BOOL
VAR_INPUT
  /// -100 to -1 = Move to HP, 1 to 100 = Move to WP, 0 = Off
  rSpeedInPercent:        REAL;
  tDelay:                 TIME;
END_VAR
END_METHOD

PROPERTY P_CurrentVal : INT
GET
END_GET
END_PROPERTY

PROPERTY P_ReadyState : BOOL
GET
END_GET
END_PROPERTY

PROPERTY P_SpeedInPercent : REAL
GET
END_GET
END_PROPERTY

END_INTERFACE

// ---- MODULE/ACTOR_VALVE/VALVE/ITF/I_VALVE_X_2.TcIO
INTERFACE I_VALVE_X_2 EXTENDS I_GENERAL_OBJECT

METHOD M_Reset : BOOL
VAR_INPUT
END_VAR
END_METHOD

METHOD M_SetReady : BOOL
VAR_INPUT
END_VAR
END_METHOD

METHOD M_ToHP : BOOL
VAR_INPUT
  tDelay:         TIME;
END_VAR
END_METHOD

METHOD M_ToWP1 : BOOL
VAR_INPUT
  tDelay:         TIME;
END_VAR
END_METHOD

PROPERTY P_InHP : BOOL
GET
END_GET
END_PROPERTY

PROPERTY P_InWP1 : BOOL
GET
END_GET
END_PROPERTY

PROPERTY P_ReadyState : BOOL
GET
END_GET
END_PROPERTY

END_INTERFACE

// ---- MODULE/ACTOR_VALVE/VALVE/ITF/I_VALVE_X_3.TcIO
INTERFACE I_VALVE_X_3 EXTENDS I_VALVE_X_2

METHOD M_SetReady : BOOL
VAR_INPUT
END_VAR
END_METHOD

METHOD M_ToWP2 : BOOL
VAR_INPUT
  tDelay:        TIME;
END_VAR
END_METHOD

PROPERTY P_InWP2 : BOOL
GET
END_GET
END_PROPERTY

END_INTERFACE

// ---- MODULE/BYTES_TO_WORD/ITF/I_WORD_TO_BYTES.TcIO
INTERFACE I_WORD_TO_BYTES EXTENDS I_GENERAL_OBJECT

PROPERTY P_VALUE : LREAL
GET
END_GET
SET
END_SET
END_PROPERTY

PROPERTY P_X_MAX : LREAL
GET
END_GET
SET
END_SET
END_PROPERTY

PROPERTY P_X_MIN : LREAL
GET
END_GET
SET
END_SET
END_PROPERTY

PROPERTY P_Y_MAX : LREAL
GET
END_GET
SET
END_SET
END_PROPERTY

PROPERTY P_Y_MIN : LREAL
GET
END_GET
SET
END_SET
END_PROPERTY

END_INTERFACE

// ---- MODULE/DATABASE/ITF/I_DATABASE.TcIO
INTERFACE I_DATABASE EXTENDS I_GENERAL_OBJECT

METHOD M_ClearTable : BOOL
VAR_INPUT
  /// Indicates the ID of the database to be used.
  udiDBID:          UDINT;
  /// Name of the table to be created.
  sTableName:       T_MaxString;
END_VAR
END_METHOD

METHOD M_Connect : BOOL
VAR_INPUT
  /// Indicates the ID of the database to be used.
  udiDBID:                  UDINT;
END_VAR
END_METHOD

METHOD M_CreateDatabase : BOOL
VAR_INPUT
  /// Address of the database configuration structure
  pDatabaseConfig:  POINTER TO BYTE;
  /// Length of the database configuration structure
  cbDatabaseConfig: UDINT;
  /// Indicates whether the newly created database should be entered as new configuration entry in the XML file.
  bCreateXMLConfig: BOOL;
  /// Returns the hDBID if/when a new configuration entry was created.
  pDBID:            POINTER TO UDINT;
END_VAR
END_METHOD

METHOD M_CreateTable : BOOL
VAR_INPUT
  /// Indicates the ID of the database to be used.
  udiDBID:                    UDINT;
  /// Name of the table that is to be read.
  sTableName:                 T_MaxString;
  /// Indicates the pointer address of the table structure array. The individual columns are written in this array.
  pTableCfg:                  POINTER TO ARRAY[0..MAX_DBCOLUMNS] OF ST_ColumnInfo;
  /// Indicates the length of the array in which the columns are configured.
  cbTableCfg:                 UDINT;
END_VAR
END_METHOD

METHOD M_DeleteTable : BOOL
VAR_INPUT
  /// Indicates the ID of the database to be used.
  udiDBID:          UDINT;
  /// Name of the table that is to be read.
  sTableName:       T_MaxString;
END_VAR
END_METHOD

METHOD M_Disconnect : BOOL
VAR_INPUT
END_VAR
END_METHOD

METHOD M_ExecuteCmd : BOOL
VAR_INPUT
  /// Indicates the ID of the database to be used.
  udiDBID:      UDINT;
  /// Addres of the command
  pExpression:  POINTER TO BYTE;
  /// Indicates the number of command.
  cbExpression: UDINT;
  /// Address of the structure array into which the records are to be written.
  pData:        POINTER TO BYTE;
  /// Indicates the size of the structure array in bytes.
  cbData:       UDINT;
  /// Address of the structure array.
  pParameter:   POINTER TO ARRAY[0..MAX_DBCOLUMNS] OF ST_ExpParameter;
  /// Indicates the size of the parameter.
  cbParameter:  UDINT; 
END_VAR
END_METHOD

METHOD M_ExecuteSimplifyCmd : BOOL
VAR_INPUT
  /// Indicates the ID of the database to be used.
  udiDBID:      UDINT;
  /// Indicates the pointer address of a string variable with the SQL command to be executed.
  pSQLCmd:      POINTER TO BYTE;
  /// Indicates the length of a SQL command to be executed.
  cbSQLCmd:     UDINT;
END_VAR
END_METHOD

METHOD M_Overwrite : BOOL
VAR_INPUT
  /// Indicates the ID of the database to be used.
  udiDBID:                    UDINT;
  /// Name of the table that is to be read.
  sTableName:                 T_MaxString;
  /// Column name of the data to be updated
  sColumnNameToUpdate:        STRING;
  /// Column value of the data to be updated
  sColumnValToUpdate:         STRING;
  /// Column name to set
  sColumnNameToSet:           STRING;
  /// New value
  sNewVal:                    STRING;
END_VAR
END_METHOD

METHOD M_Read : BOOL
VAR_INPUT
  /// Indicates the ID of the database to be used.
  udiDBID:                    UDINT;
  /// Name of the table that is to be read.
  sTableName:                 T_MaxString;
  /// Symbol name to be read from the standard table structure.
  sDBSymbolName:              STRING;
  /// Sorting column (ID, timestamp, name or value)
  eOrderBy:                   E_OrderColumn;
  /// Sorting direction (ASC or DESC)
  eOrderType:                 E_OrderType;
  /// Indicates the index of the first record to be read.
  nStartIndex:                UDINT;
  /// Indicates the number of records to be read.
  nRecordCount:               UDINT;
  /// Address of the structure array into which the records are to be written.
  pData2:                     POINTER TO ST_StandardRecord;
  /// Indicates the size of the structure array in bytes.
  cbData:                     UDINT;
END_VAR
END_METHOD

METHOD M_ReadStruct : BOOL
VAR_INPUT
  /// Indicates the ID of the database to be used.
  udiDBID:                    UDINT;
  /// Name of the table that is to be read.
  sTableName:                 T_MaxString;
  /// Address of the array containing the column name to be read.
  pColumnNames:               POINTER TO ARRAY [0..MAX_DBCOLUMNS] OF STRING(50);
  /// Length of the column name array
  cbColumnNames:              UDINT;
  /// Name the sorting column
  sOrderByColumn:             STRING(50);
  /// Sorting direction (ASC or DESC)
  eOrderType:                 E_OrderType;
  /// Indicates the index of the first record to be read.
  nStartIndex:                UDINT;
  /// Indicates the number of records to be read.
  nRecordCount:               UDINT;
  /// Address of the structure array into which the records are to be written.
  pData:                      POINTER TO BYTE;
  /// Indicates the size of the structure array in bytes.
  cbData:                     UDINT;
END_VAR
END_METHOD

METHOD M_Reset : BOOL
VAR_INPUT
END_VAR
END_METHOD

METHOD M_SetReady : BOOL
VAR_INPUT
END_VAR
END_METHOD

METHOD M_TableExistCheck : BOOL
VAR_INPUT
  /// Indicates the ID of the database to be used.
  udiDBID:                    UDINT;
  /// Name of the table that is to be read.
  sTableName:                 T_MaxString;
END_VAR
VAR_OUTPUT
  /// Result
  bResult:                    BOOL;
END_VAR
END_METHOD

METHOD M_Write : BOOL
VAR_INPUT
  /// Indicates the ID of the database to be used.
  udiDBID:            UDINT;
  /// Name of the table that is to be write.
  sTableName:         T_MaxString;
  /// Address of the variable to be logged in the standard table structure.
  pValue:             POINTER TO BYTE;
  /// Length of the variable to be logged.
  cbValue:            UDINT;
  /// Name that is logged in the table.
  sDBSymbolName:      STRING;
  /// Indicates the write mode. (append, update, ring buffer)
  eDBWriteMode:       E_WriteMode;
  /// Additional parameter(s) for the "ring buffer" write mode.
  nRingBuffParameter: UDINT;
END_VAR
END_METHOD

METHOD M_WriteBySymbol : BOOL
VAR_INput
  /// Indicates the ID of the database to be used.
  udiDBID:            UDINT;
  /// Name of the table that is to be write.
  sTableName:         T_MaxString;
  /// ADS device from which a symbol is to be logged in the standard table structure.
  stADSDevice: ST_ADSDevice;
  /// Symbol name of the variable to be written
  stSymbol: ST_Symbol;
  /// Indicates the write mode. (append, update, ring buffer)
  eDBWriteMode:       E_WriteMode;
  /// Additional parameter(s) for the "ring buffer" write mode.
  nRingBuffParameter: UDINT;
END_VAR
END_METHOD

METHOD M_WriteStruct : BOOL
VAR_INPUT
  /// Indicates the ID of the database to be used.
  udiDBID:        UDINT;
  /// Name of the table that is to be write.
  sTableName:     T_MaxString;
  /// Address of a structure that is to be logged in a freely selectable table structure.
  pRecord:        POINTER TO BYTE;
  /// Length of the structure to be written
  cbRecord:       UDINT;
  /// Address of the array containing the column name to be filled.
  pColumnNames:   POINTER TO ARRAY [0..MAX_DBCOLUMNS] OF STRING(50);
  /// Length of the column name array
  cbColumnNames:  UDINT;
END_VAR
END_METHOD

PROPERTY P_Connected : BOOL
GET
END_GET
END_PROPERTY

PROPERTY P_Error : BOOL
GET
END_GET
END_PROPERTY

END_INTERFACE

// ---- MODULE/DATABASE/ITF/I_INFLUXDB_ADS.TcIO
INTERFACE I_INFLUXDB_ADS EXTENDS I_GENERAL_OBJECT

METHOD M_BucketExistCheck : BOOL
VAR_INPUT
  /// Name of the table that is to be read.
  sBucketName:                T_MaxString;
END_VAR
VAR_OUTPUT
  /// Result
  bResult:                    BOOL;
END_VAR
END_METHOD

METHOD M_ClearMeasurement : BOOL
VAR_INPUT
  /// Bucket name
  sBucketName:          T_MaxString;
  /// Name of the measure to clear
  sMeasurementName:     T_MaxString;
  /// From date time (Range)
  dtFrom:               DT;
  /// To date time (Range)
  dtTo:                 DT;
END_VAR
VAR_OUTPUT
	/// Result
	bResult	: BOOL;
END_VAR
END_METHOD

METHOD M_DeleteAllMeasurements : BOOL
VAR_INPUT
  /// Bucket name
  sBucketName:          T_MaxString;
END_VAR
VAR_OUTPUT
	/// Result
	bResult	: BOOL;
END_VAR
END_METHOD

METHOD M_DeleteField : BOOL
VAR_INPUT
  /// Bucket name
  sBucketName:          T_MaxString;
  /// Measurement Name
  sMeasurementName:     T_MaxString;
  /// Tag Name
  sTagName:             T_MaxString;
  /// Field Name
  sFieldName:           T_MaxString;
END_VAR
VAR_OUTPUT
  /// Result
  bResult:              BOOL;
END_VAR
END_METHOD

METHOD M_DeleteMeasurement : BOOL
VAR_INPUT
  /// Bucket name
  sBucketName:          T_MaxString;
  /// Name of the measure to delete.
  sMeasurementName:     T_MaxString;
END_VAR
VAR_OUTPUT
	/// Result
	bResult	: BOOL;
END_VAR
END_METHOD

METHOD M_DeleteTag : BOOL
VAR_INPUT
  /// Bucket name
  sBucketName:          T_MaxString;
  /// Measurement Name
  sMeasurementName:     T_MaxString;
  /// Tag Name
  sTagName:             T_MaxString;
END_VAR
VAR_OUTPUT
  /// Result
  bResult:              BOOL;
END_VAR
END_METHOD

METHOD M_DeleteTagContentBlock : BOOL
VAR_INPUT
  /// Bucket name
  sBucketName:          T_MaxString;
  /// Measurement Name
  sMeasurementName:     T_MaxString;
  /// Tag Name
  sTagName:             T_MaxString;
  /// Date and time from
  dtFrom:               DT;
  /// Date and Time to
  dtTo:                 DT;
END_VAR
VAR_OUTPUT
  /// Result
  bResult:              BOOL;
END_VAR
END_METHOD

METHOD M_FieldExistCheck : BOOL
VAR_INPUT
  /// Bucket name
  sBucketName:          T_MaxString;
  /// Measurement Name
  sMeasurementName:     T_MaxString;
  /// Tag Name
  sTagName:             T_MaxString;
  /// Field Name
  sFieldName:           T_MaxString;
END_VAR
VAR_OUTPUT
  /// Result
  bResult:              BOOL;
END_VAR
END_METHOD

METHOD M_GetTotalMeasurements : BOOL
VAR_INPUT
  /// Bucket name
  sBucketName:          T_MaxString;
END_VAR
VAR_OUTPUT
  /// Process success
  bResult:              BOOL;
  /// Result value
  uiResult:             UINT;
END_VAR
END_METHOD

METHOD M_MeasurementExistCheck : BOOL
VAR_INPUT
  /// Bucket name
  sBucketName:          T_MaxString;
  /// Name of the table that is to be read.
  sMeasurementName:     T_MaxString;
END_VAR
VAR_OUTPUT
  /// Result
  bResult:              BOOL;
END_VAR
END_METHOD

METHOD M_Reset : BOOL
VAR_INPUT
END_VAR
END_METHOD

METHOD M_SetReady : BOOL
VAR_INPUT
END_VAR
END_METHOD

METHOD M_TagExistCheck : BOOL
VAR_INPUT
  /// Bucket name
  sBucketName:          T_MaxString;
  /// Measurement Name
  sMeasurementName:     T_MaxString;
  /// Tag Name
  sTagName:             T_MaxString;
END_VAR
VAR_OUTPUT
  /// Result
  bResult:              BOOL;
END_VAR
END_METHOD

METHOD M_WriteStruct : BOOL
VAR_INPUT
  /// Bucket name
	sBucketName:                  T_MaxString;
	/// Name of the table that is to be read.
	sMeasurementName:             T_MaxString;
	/// Tag name
	sTagName:                     T_MaxString;
  /// Field values list
	stFieldValues:                ST_DATABASE_RECORD;
  /// Field struct content (Variable names)
  //pFieldStructContent:        POINTER TO ARRAY [0..99] OF T_MaxString;
	/// Field names list: names that appear in the database
	//pFieldNames:                POINTER TO ARRAY [0..99] OF T_MaxString;
END_VAR
VAR_OUTPUT
	/// Result
	bResult	: BOOL;
END_VAR
END_METHOD

PROPERTY P_ADSLifeBit : BOOL
GET
END_GET
END_PROPERTY

PROPERTY P_ADSState : BOOL
GET
END_GET
END_PROPERTY

PROPERTY P_Connected : BOOL
GET
END_GET
END_PROPERTY

PROPERTY P_Error : BOOL
GET
END_GET
END_PROPERTY

PROPERTY P_InfluxDBLifeBit : BOOL
GET
END_GET
END_PROPERTY

PROPERTY P_InfluxDBState : BOOL
GET
END_GET
END_PROPERTY

END_INTERFACE

// ---- MODULE/FREQUENCE/ITF/I_FREQ_GEN.TcIO
INTERFACE I_FREQ_GEN EXTENDS I_GENERAL_OBJECT

METHOD M_SetFrequence : bool
VAR_INPUT
	iFreqence: INT;
END_VAR
END_METHOD

PROPERTY P_FTrig : BOOL
GET
END_GET
END_PROPERTY

PROPERTY P_RTrig : BOOL
GET
END_GET
END_PROPERTY

PROPERTY P_State : BOOL
GET
END_GET
END_PROPERTY

END_INTERFACE

// ---- MODULE/GENERAL/INPUTS/ITF/I_BINARY_SWITCH_SENS.TcIO
INTERFACE I_BINARY_SWITCH_SENS EXTENDS I_BINARY_SWITCH

METHOD M_START_SENS : BOOL
VAR_INPUT
	bState: BOOL;
	tDelay: TIME;
	eEventType: ENUM_EVENT_TYPE;
END_VAR
END_METHOD

METHOD M_STOP_SENS : BOOL
VAR_INPUT
END_VAR
END_METHOD

PROPERTY P_STATE_SENS : BOOL
GET
END_GET
END_PROPERTY

END_INTERFACE

// ---- MODULE/GENERAL/SIMU_ANALOG_IN/I_SIMU_ANALOG_IN.TcIO
INTERFACE I_SIMU_ANALOG_IN EXTENDS I_ANALOG_IN

PROPERTY P_SETPOINT : LREAL
SET
END_SET
END_PROPERTY

END_INTERFACE

// ---- MODULE/HMI/ITF/I_HMI_CTRL.TcIO
INTERFACE I_HMI_CTRL EXTENDS I_GENERAL_OBJECT

METHOD M_CloseHMI : BOOL
VAR_INPUT
END_VAR
END_METHOD

METHOD M_HideWinKeyboard : BOOL
VAR_INPUT
END_VAR
END_METHOD

METHOD M_PCReboot : BOOL
VAR_INPUT
END_VAR
END_METHOD

METHOD M_PCShutdown : BOOL
VAR_INPUT
END_VAR
END_METHOD

METHOD M_SetReady : BOOL
VAR_INPUT
END_VAR
END_METHOD

METHOD M_ShowWinKeyboard : BOOL
VAR_INPUT
END_VAR
END_METHOD

METHOD M_StartHMI : BOOL
VAR_INPUT
END_VAR
END_METHOD

END_INTERFACE

// ---- MODULE/SAFETY/ITF/I_ESTOP.TcIO
INTERFACE I_ESTOP	EXTENDS I_GENERAL_OBJECT

METHOD M_Quit : BOOL
VAR_INPUT
END_VAR
END_METHOD

METHOD M_Reset : BOOL
VAR_INPUT
END_VAR
END_METHOD

PROPERTY P_E_StopAktiv : BOOL
GET
END_GET
END_PROPERTY

PROPERTY P_E_StopLoadingLeftAktiv : BOOL
GET
END_GET
END_PROPERTY

PROPERTY P_E_StopLoadingRightAktiv : BOOL
GET
END_GET
END_PROPERTY

PROPERTY P_E_StopQuittieren : BOOL
GET
END_GET
END_PROPERTY

PROPERTY P_E_StopWeighSideAktiv : BOOL
GET
END_GET
END_PROPERTY

END_INTERFACE

// ---- MODULE/TRAFFIC_LIGHT/ITFs/I_TrafficLight.TcIO
INTERFACE I_TrafficLight

METHOD M_Beep : BOOL
VAR_INPUT
	/// On/Off signal
	bEnable:				BOOL;
	/// Flashing frequency (0 = Permanently On, 1 = 1s alternately, ...)
	uiBlinkFrequency:		UINT;
END_VAR
END_METHOD

METHOD M_Green : BOOL
VAR_INPUT
	/// On/Off light
	bEnable:				BOOL;
	/// Flashing frequency (0 = Permanently On, 1 = 1s alternately, ...)
	uiBlinkFrequency:		UINT;
	/// Reset all colors, before set this color
	bResetOther:			BOOL;
END_VAR
END_METHOD

METHOD M_Multicolor : BOOL
VAR_INPUT
	/// Enable green
	bGreen:					BOOL;
	/// Enable yellow
	bYellow:				BOOL;
	/// Enable red
	bRed:					BOOL;
	/// Flashing frequency (0 = Permanently On, 1 = 1s alternately, ...)
	uiBlinkFrequency:		UINT;
END_VAR
END_METHOD

METHOD M_Red : BOOL
VAR_INPUT
	/// On/Off light
	bEnable:				BOOL;
	/// Flashing frequency (0 = Permanently On, 1 = 1s alternately, ...)
	uiBlinkFrequency:		UINT;
	/// Reset all colors, before set this color
	bResetOther:			BOOL;
END_VAR
END_METHOD

METHOD M_Reset : BOOL
VAR_INPUT
END_VAR
END_METHOD

METHOD M_Yellow : BOOL
VAR_INPUT
	/// On/Off light
	bEnable:				BOOL;
	/// Flashing frequency (0 = Permanently On, 1 = 1s alternately, ...)
	uiBlinkFrequency:		UINT;
	/// Reset all colors, before set this color
	bResetOther:			BOOL;
END_VAR
END_METHOD

PROPERTY P_BeepState : BOOL
GET
END_GET
END_PROPERTY

PROPERTY P_GreenState : BOOL
GET
END_GET
END_PROPERTY

PROPERTY P_RedState : BOOL
GET
END_GET
END_PROPERTY

PROPERTY P_YellowState : BOOL
GET
END_GET
END_PROPERTY

END_INTERFACE

// ---- ORGANISATION/DATE_TIME/ITF/I_CLOCK.TcIO
INTERFACE I_CLOCK EXTENDS I_GENERAL_OBJECT

METHOD M_GetTimerET : STRING
VAR_INPUT
  /// Default: hhh:mm:ss
  bCustomFormat:      BOOL;
  /// Timeformat: mm/ss or hh-mm-ss or dd/hh/mm/ss
  sFormat:            STRING;
END_VAR
END_METHOD

METHOD M_PauseTimer : BOOL
VAR_INPUT
END_VAR
END_METHOD

METHOD M_StartTimer : BOOL
VAR_INPUT
END_VAR
END_METHOD

METHOD M_StopTimer : BOOL
VAR_INPUT
END_VAR
END_METHOD

METHOD M_WaitForTimer : BOOL
VAR_INPUT
END_VAR
END_METHOD

PROPERTY P_SystemTime : STRING
GET
END_GET
END_PROPERTY

END_INTERFACE

// ---- ORGANISATION/EVENT_LOGGER/ITFs/I_EVENT_LOGGER.TcIO
INTERFACE I_EVENT_LOGGER EXTENDS I_GENERAL_OBJECT

METHOD M_ErrorMsg : BOOL
VAR_INPUT
  udiID:                        UDINT;
  sMsg:                         T_MaxString;
  bWithConfirmation:            BOOL;
END_VAR
END_METHOD

METHOD M_InfoMsg : BOOL
VAR_INPUT
  udiID:                   UDINT;
  sMsg:                    T_MaxString;
END_VAR
END_METHOD

METHOD M_WarningMsg : BOOL
VAR_INPUT
  udiID:                   UDINT;
  sMsg:                    T_MaxString;
END_VAR
END_METHOD

END_INTERFACE

// ---- ORGANISATION/GENERAL/ITF/I_FunctionCtrl.TcIO
INTERFACE I_FunctionCtrl

PROPERTY Busy : BOOL
GET
END_GET
END_PROPERTY

PROPERTY Done : BOOL
GET
END_GET
END_PROPERTY

PROPERTY Error : BOOL
GET
END_GET
END_PROPERTY

PROPERTY ErrorCode : WORD
GET
END_GET
END_PROPERTY

METHOD Execute : BOOL
VAR_INPUT
END_VAR
END_METHOD

PROPERTY Ready : BOOL
GET
END_GET
END_PROPERTY

METHOD Reset : BOOL
VAR_INPUT
END_VAR
END_METHOD

END_INTERFACE

// ---- ORGANISATION/GENERAL/ITF/I_GENERAL.TcIO
INTERFACE I_GENERAL

METHOD M_CyclicRun : BOOL
VAR_INPUT
END_VAR
END_METHOD

PROPERTY P_ObjectID : STRING
GET
END_GET
SET
END_SET
END_PROPERTY

END_INTERFACE

// ---- ORGANISATION/OP_MODE/ITF/I_OP_MODE.TcIO
INTERFACE I_OP_MODE

METHOD M_AUTOMATIC
VAR_INPUT
END_VAR
END_METHOD

METHOD M_DEBUG
VAR_INPUT
END_VAR
END_METHOD

METHOD M_MANUAL
VAR_INPUT
END_VAR
END_METHOD

METHOD M_OP_MODE_OFF
VAR_INPUT
END_VAR
END_METHOD

METHOD M_OP_MODE_ON : BOOL
VAR_INPUT
END_VAR
END_METHOD

METHOD M_RESET : BOOL
VAR_INPUT
END_VAR
END_METHOD

PROPERTY P_CONTROL_ON : bool
GET
END_GET
SET
END_SET
END_PROPERTY

PROPERTY P_EMERGANCY_STOP : bool
GET
END_GET
SET
END_SET
END_PROPERTY

PROPERTY P_INIT_OK : BOOL
GET
END_GET
SET
END_SET
END_PROPERTY

PROPERTY P_OP_MODE_STATE : INT
GET
END_GET
END_PROPERTY

PROPERTY P_QUIT : BOOL
GET
END_GET
END_PROPERTY

END_INTERFACE

// ---- ORGANISATION/OP_MODE/ITF/I_OP_MODE_PAUSE.TcIO
INTERFACE I_OP_MODE_PAUSE EXTENDS I_OP_MODE

METHOD M_OP_MODE_TO_PAUSE
VAR_INPUT
END_VAR
END_METHOD

PROPERTY P_PAUSE_ACTIVATE : BOOL
GET
END_GET
END_PROPERTY

END_INTERFACE

// ---- ORGANISATION/OP_MODE/ITF/I_OP_MODE_PAUSE_VISU.TcIO
INTERFACE I_OP_MODE_PAUSE_VISU EXTENDS I_GENERAL_OBJECT

METHOD M_ResetModeSelection : BOOL
VAR_INPUT
END_VAR
END_METHOD

PROPERTY P_BreakPressureDetSelected : BOOL
GET
END_GET
END_PROPERTY

PROPERTY P_EnduranceRunSelected : BOOL
GET
END_GET
END_PROPERTY

PROPERTY P_HandSelected : BOOL
GET
END_GET
END_PROPERTY

PROPERTY P_JogCounterCyl1_Active : BOOL
GET
END_GET
END_PROPERTY

PROPERTY P_JogCounterCyl2_Active : BOOL
GET
END_GET
END_PROPERTY

PROPERTY P_JogCounterCyl3_Active : BOOL
GET
END_GET
END_PROPERTY

PROPERTY P_JogCounterCyl4_Active : BOOL
GET
END_GET
END_PROPERTY

PROPERTY P_JogSelected : BOOL
GET
END_GET
END_PROPERTY

PROPERTY P_LeakTest1Selected : BOOL
GET
END_GET
END_PROPERTY

PROPERTY P_LeakTest2Selected : BOOL
GET
END_GET
END_PROPERTY

END_INTERFACE

// ---- SUBSTATION/STATION_NEST/ITF/I_PROCESS_MAIN.TcIO
INTERFACE I_PROCESS_MAIN EXTENDS I_GENERAL_OBJECT

METHOD M_BreakPressureDet : BOOL
VAR_INPUT
  stBreakPressureParams:                 ST_RECIPE_BREAK_PRESSURE;
END_VAR
END_METHOD

METHOD M_EnduranceRun : BOOL
VAR_INPUT
  stEnduranceRunParams:                 ST_RECIPE_ENDURANCE_RUN;
END_VAR
END_METHOD

METHOD M_EStop : BOOL
VAR_INPUT
END_VAR
END_METHOD

METHOD M_LeakTest1 : BOOL
VAR_INPUT
  stLeakTest1Params:                 ST_RECIPE_LEAK_TEST1;
END_VAR
END_METHOD

METHOD M_LeakTest2 : BOOL
VAR_INPUT
  stLeakTest2Params:                 ST_RECIPE_LEAK_TEST2;
END_VAR
END_METHOD

METHOD M_Reset : BOOL
VAR_INPUT
END_VAR
END_METHOD

METHOD M_SetReady : BOOL
VAR_INPUT
END_VAR
END_METHOD

METHOD M_Stop : BOOL
END_METHOD

METHOD M_StopEngine : BOOL
VAR_INPUT
END_VAR
END_METHOD

PROPERTY P_CurrentCycleNest1 : UDINT
GET
END_GET
END_PROPERTY

PROPERTY P_CurrentCycleNest2 : UDINT
GET
END_GET
END_PROPERTY

PROPERTY P_CurrentCycleNest3 : UDINT
GET
END_GET
END_PROPERTY

PROPERTY P_CurrentCycleNest4 : UDINT
GET
END_GET
END_PROPERTY

PROPERTY P_ReadyState : BOOL
GET
END_GET
END_PROPERTY

END_INTERFACE

// ---- SUBSTATION/STATION_NEST/ITF/I_PROCESS_NEST1.TcIO
INTERFACE I_PROCESS_NEST1 EXTENDS I_PROCESS_NEST2_4

METHOD M_BreakPressureDet : BOOL
VAR_INPUT
  stBreakPressureParams:                ST_RECIPE_BREAK_PRESSURE;
END_VAR
END_METHOD

METHOD M_LeakTest2 : BOOL
VAR_INPUT
  stLeakTest2Params:                 ST_RECIPE_LEAK_TEST2;
END_VAR
END_METHOD

METHOD M_MaxSpeedRecord : BOOL
VAR_INPUT
  stEnduranceRunParams:                 ST_RECIPE_ENDURANCE_RUN;
END_VAR
END_METHOD

METHOD M_MoveTestCyl1ToHP : BOOL
VAR_INPUT
  rWorkForceA:                    REAL;
  rWorkForceB:                    REAL;
  rLoadForceA:                    REAL;
  rLoadForceB:                    REAL;
END_VAR
END_METHOD

PROPERTY P_MaxSpeedInMmPerSHP : REAL
GET
END_GET
END_PROPERTY

PROPERTY P_MaxSpeedInMmPerSWP : REAL
GET
END_GET
END_PROPERTY

PROPERTY P_ReadyState : BOOL
GET
END_GET
END_PROPERTY

PROPERTY P_SpeedEfficiencyFactor : REAL
GET
END_GET
END_PROPERTY

END_INTERFACE

// ---- SUBSTATION/STATION_NEST/ITF/I_PROCESS_NEST2_4.TcIO
INTERFACE I_PROCESS_NEST2_4 EXTENDS I_GENERAL_OBJECT

METHOD M_EnduranceRun : BOOL
VAR_INPUT
  udiCycles:                            UDINT;
  stEnduranceRunParams:                 ST_RECIPE_ENDURANCE_RUN;
END_VAR
END_METHOD

METHOD M_LeakTest1 : BOOL
VAR_INPUT
  stLeakTest1Params:                 ST_RECIPE_LEAK_TEST1;
END_VAR
END_METHOD

METHOD M_MeasureStrokeLength : BOOL
VAR_INPUT
  bCylinderDecoupled:             BOOL;
  rWorkForceA:                    REAL;
  rWorkForceB:                    REAL;
  rLoadForceA:                    REAL;
  rLoadForceB:                    REAL;
END_VAR
END_METHOD

METHOD M_MoveToSetPos : BOOL
VAR_INPUT
END_VAR
END_METHOD

METHOD M_Reset : BOOL
VAR_INPUT
END_VAR
END_METHOD

METHOD M_ResetDistance : BOOL
VAR_INPUT
END_VAR
END_METHOD

METHOD M_SetEnableState : BOOL
VAR_INPUT
  bEnable:              BOOL;
END_VAR
END_METHOD

METHOD M_SetReady : BOOL
VAR_INPUT
END_VAR
END_METHOD

METHOD M_Stop : BOOL
END_METHOD

METHOD M_StopEngine : BOOL
VAR_INPUT
END_VAR
END_METHOD

METHOD M_VentCylinder : BOOL
VAR_INPUT
  bCylinderDecoupled:             BOOL;
  uiVentCount:                    UINT;
  rWorkForceA:                    REAL;
  rWorkForceB:                    REAL;
  rLoadForceA:                    REAL;
  rLoadForceB:                    REAL;
END_VAR
END_METHOD

PROPERTY P_CurrentCycle : UDINT
GET
END_GET
END_PROPERTY

PROPERTY P_EnableState : BOOL
GET
END_GET
END_PROPERTY

PROPERTY P_NokDifference : REAL
GET
END_GET
END_PROPERTY

PROPERTY P_NokLimitInPercent : UINT
GET
END_GET
END_PROPERTY

PROPERTY P_ReadyState : BOOL
GET
END_GET
END_PROPERTY

PROPERTY P_SerialNr : STRING
GET
END_GET
SET
END_SET
END_PROPERTY

PROPERTY P_Timer : STRING
GET
END_GET
END_PROPERTY

END_INTERFACE

// ---- PROGRAMS/PrgMeasure.TcPOU
PROGRAM PrgMeasure
VAR_INPUT
  bRecord:                                                    BOOL;
END_VAR
VAR
  uiSeq:                                                      UINT := 0;
  i:                                                          UINT;
END_VAR
VAR // Time
  fbLocalSystemTime:                                          FB_LocalSystemTime := ( bEnable := TRUE, dwCycle := 1 );
  systemTime:                                                 TIMESTRUCT;
  sCurrentDateTime:                                           STRING;
END_VAR
VAR // TwincatADSGateway parameter
  bLifeBit:                                                   BOOL;
  bAdsConnected:                                              BOOL;
  bReady:                                                     BOOL;
  bBusy:                                                      BOOL;
  bResult:                                                    BOOL;
  bOpenKeyboard:                                              BOOL;
  bCloseHMI:                                                  BOOL;
  bShutdownPc:                                                BOOL;
  bRestartPc:                                                 BOOL;
  sLog:                                                       T_MaxString;
  stFieldValues:                                              ST_DATABASE_RECORD;
  arrFieldStructContent:                                      ARRAY [0..99] OF T_MaxString;
  arrFieldNames:                                              ARRAY [0..99] OF T_MaxString;
  liFreeSpaceOnC:                                             LINT;
  fbInfluxDB:                                                 FB_INFLUX_DB_ADS(itfOpMode:= PrgOrg.fbOpMode,
                                                                               itfEventLogger:= PrgOrg.fbEventLogger);
END_VAR
VAR // Params from DB Settings
  sMeasurementNameFromCfg:                                    T_MaxString;
  sTagNameFromCfg:                                            T_MaxString;
  uiTagNameIDFromCfg:                                         UINT;
  bCheckMesurementExistSelected:                              BOOL;
  bCheckTagExistSelected:                                     BOOL;
  dtFromFromCfg:                                              DT := DT#2024-01-01-00:00:00;
  dtToFromCfg:                                                DT := DT#2024-01-01-00:00:00;
  bDeleteAllTagContentChecked:                                BOOL;
  sTest:                                                      STRING;
END_VAR
VAR // Get total measurements
  uiTotalMeasurementsSeq:                                     UINT := 0;
  uiTotalMeasurements:                                        UINT;
  bGetTotalMeasurements:                                      BOOL;
  bGetTotalMeasurementsProcessSuccess:                        BOOL;
END_VAR
VAR // Measurement exist
  uiMeasurementExistSeq:                                      UINT := 0;
  bGetMeasurementExist:                                       BOOL;
  bMeasurementExist:                                          BOOL;
END_VAR
VAR // Tag exist
  uiTagExistSeq:                                              UINT := 0;
  bGetTagExist:                                               BOOL;
  bTagExist:                                                  BOOL;
END_VAR
VAR // Delete measurement
  uiDeleteMeasurementSeq:                                     UINT := 0;
  bDeleteMeasurement:                                         BOOL;
  bDeleteMeasurementResult:                                   BOOL;
END_VAR
VAR // Delete Tag
  uiDeleteTagSeq:                                             UINT := 0;
  bDeleteTag:                                                 BOOL;
  bDeleteTagResult:                                           BOOL;
END_VAR
VAR // Delete Tag content block
  uiDeleteTagContentBlockSeq:                                 UINT := 0;
  bDeleteTagContentBlock:                                     BOOL;
  bDeleteTagContentBlockResult:                               BOOL;
END_VAR
VAR // Timer
  iSaveSeq:                                                   INT := 0;
  iSeqCounter:                                                INT := 1;
  bSaveTrigger:                                               BOOL;
  bSaveBusy:                                                  BOOL;
  tInterval:                                                  TIME := T#500MS;
  tonInterval:                                                TON;
  tSwitchTime:                                                TIME := T#10H;
  tonSwitchTimer:                                             TON;
  tFailedSaveLimitTime:                                       TIME := T#7M;
  tonFailedSavelimitTimer:                                    TON;
  uiAllowedSaveFail:                                          UINT := 3;
END_VAR
VAR // Params
  sBucketName:                                                T_MaxString := '3925-HZP';
  sMeasurementName:                                           T_MaxString := 'Artikel';
  sTagName:                                                   T_MaxString := 'Dauerlauf777';
  bSaveSuccess:                                               BOOL;
  uiFailedSaveCounter:                                        UINT := 0;
  
  liTargetCycles:                                             LINT;
  rTargetTestPressureInBarA:                                  REAL;
  rTargetTestPressureInBarB:                                  REAL;
  rTargetTestForceInKNA:                                      REAL;
  rTargetTestForceInKNB:                                      REAL;
  rTargetCounterPressureInBarA:                               REAL;
  rTargetCounterPressureInBarB:                               REAL;
  rTargetCounterForceInKNA:                                   REAL;
  rTargetCounterForceInKNB:                                   REAL;
  rTargetSpeedAInMmPerS:                                      REAL;
  rTargetSpeedBInMmPerS:                                      REAL;
  lrNokLimit:                                                 LREAL;
END_VAR

(* Actions *)
A_000_FBs();
A_010_DBInit();
A_100_SaveToDB();
A_110_TotalMeasurements();
A_120_MeasurementExistCheck();
A_130_TagExistCheck();
A_140_DeleteMeasurement();
A_150_DeleteTag();
A_160_DeleteTagContentBlock();

sTest := TO_STRING(dtFromFromCfg);

ACTION A_000_FBs:
(* FBs *)
fbLocalSystemTime(systemTime=> systemTime);
fbInfluxDB(bResult:= bResult,
           bADSLifeBit:= bLifeBit,
           bAdsConnected:= bAdsConnected,
           bReady:= bReady,
           bBusy:= bBusy);
END_ACTION

ACTION A_010_DBInit:
(* Define struct content names *)
// assign variable names to struct content list
arrFieldStructContent[0] := 'sTimeStamp';
arrFieldStructContent[1] := 'sTimer';
arrFieldStructContent[2] := 'liTargetCycles';
arrFieldStructContent[3] := 'liActiveCycle';
arrFieldStructContent[4] := 'iTestDirection';
arrFieldStructContent[5] := 'rTargetTestPressureInBarA';
arrFieldStructContent[6] := 'rTargetTestPressureInBarB';
arrFieldStructContent[7] := 'rCurrentTestPressureInBar';
arrFieldStructContent[8] := 'rTargetTestForceInKNA';
arrFieldStructContent[9] := 'rTargetTestForceInKNB';
arrFieldStructContent[10] := 'rCurrentTestForceInKN';
arrFieldStructContent[11] := 'rTestPressureAInBar';
arrFieldStructContent[12] := 'rTestPressureBInBar';
arrFieldStructContent[13] := 'rBreakawayPressureInBar';
arrFieldStructContent[14] := 'rBreakawayPressureAInBar';
arrFieldStructContent[15] := 'rBreakawayPressureBInBar';
arrFieldStructContent[16] := 'rReservoirPressureInBar';
arrFieldStructContent[17] := 'rTargetCounterPressureInBarA';
arrFieldStructContent[18] := 'rTargetCounterPressureInBarB';
arrFieldStructContent[19] := 'rCurrentCounterPressureInBar';
arrFieldStructContent[20] := 'rTargetCounterForceInKNA';
arrFieldStructContent[21] := 'rTargetCounterForceInKNB';
arrFieldStructContent[22] := 'rCurrentCounterForceInKN';
arrFieldStructContent[23] := 'lrPosition';
arrFieldStructContent[24] := 'lrPositionMin';
arrFieldStructContent[25] := 'lrPositionMax';
arrFieldStructContent[26] := 'lrCylStrokeLength';
arrFieldStructContent[27] := 'lrTemperature';
arrFieldStructContent[28] := 'lrCylPistonSurfaceA';
arrFieldStructContent[29] := 'lrCylPistonSurfaceB';
arrFieldStructContent[30] := 'lrNokLimit';
arrFieldStructContent[31] := 'lrCurrentNokDifference';
arrFieldStructContent[32] := 'lrCurrentNokLimitInPercent';
arrFieldStructContent[33] := 'lrTargetSpeedAInMmPerS';
arrFieldStructContent[34] := 'lrTargetSpeedBInMmPerS';
arrFieldStructContent[35] := 'lrCurrentSpeedInMmPerS';

// assign variable names to database content
arrFieldNames[0] := 'Zeitstempel';
arrFieldNames[1] := 'Timer';
arrFieldNames[2] := 'SollZyklen';
arrFieldNames[3] := 'AktiverZyklus';
arrFieldNames[4] := 'Prüfrichtung';
arrFieldNames[5] := 'TestdruckInBarA_Soll';
arrFieldNames[6] := 'TestdruckInBarB_Soll';
arrFieldNames[7] := 'TestdruckInBar_Ist';
arrFieldNames[8] := 'TestkraftInKNA_Soll';
arrFieldNames[9] := 'TestkraftInKNB_Soll';
arrFieldNames[10] := 'TestkraftInKN_Ist';
arrFieldNames[11] := 'TestDruckAInBar';
arrFieldNames[12] := 'TestDruckBInBar';
arrFieldNames[13] := 'LosbrechdruckInBar';
arrFieldNames[14] := 'LosbrechdruckAInBar';
arrFieldNames[15] := 'LosbrechdruckBInBar';
arrFieldNames[16] := 'DruckspeicherdruckInBar';
arrFieldNames[17] := 'GegenhaltezylinderdruckInBarA_Soll';
arrFieldNames[18] := 'GegenhaltezylinderdruckInBarB_Soll';
arrFieldNames[19] := 'GegenhaltezylinderdruckInBar_Ist';
arrFieldNames[20] := 'GegenhaltezylinderkraftInKNA_Soll';
arrFieldNames[21] := 'GegenhaltezylinderkraftInKNB_Soll';
arrFieldNames[22] := 'GegenhaltezylinderkraftInKN_Ist';
arrFieldNames[23] := 'Position';
arrFieldNames[24] := 'PositionMin';
arrFieldNames[25] := 'PositionMax';
arrFieldNames[26] := 'HublängeInMm';
arrFieldNames[27] := 'TemperaturInC';
arrFieldNames[28] := 'KolbenflächeA';
arrFieldNames[29] := 'KolbenflächeB';
arrFieldNames[30] := 'NOKDifferenzLimit';
arrFieldNames[31] := 'NOKDifferenz_Ist';
arrFieldNames[32] := 'NOKDifferenzInProzent_Ist';
arrFieldNames[33] := 'GeschwindigkeitAInMmProS_Soll';
arrFieldNames[34] := 'GeschwindigkeitBInMmProS_Soll';
arrFieldNames[35] := 'GeschwindigkeitInMmProS_Ist';

// Set
IF PrgVisu.fbVisuOPMode.P_EnduranceRunSelected THEN
  sTagName := 'Dauerlauf';
  liTargetCycles := PrgStation.stRecipeParams.stRecipeEnduranceRun.udiCycles;
  rTargetTestPressureInBarA := PrgStation.stRecipeParams.stRecipeEnduranceRun.rWorkPressureA;
  rTargetTestPressureInBarB := PrgStation.stRecipeParams.stRecipeEnduranceRun.rWorkPressureB;
  rTargetTestForceInKNA := PrgStation.stRecipeParams.stRecipeEnduranceRun.rWorkForceA;
  rTargetTestForceInKNB := PrgStation.stRecipeParams.stRecipeEnduranceRun.rWorkForceB;
  rTargetCounterPressureInBarA := PrgStation.stRecipeParams.stRecipeEnduranceRun.rLoadPressureA;
  rTargetCounterPressureInBarB := PrgStation.stRecipeParams.stRecipeEnduranceRun.rLoadPressureB;
  rTargetCounterForceInKNA := PrgStation.stRecipeParams.stRecipeEnduranceRun.rLoadForceA;
  rTargetCounterForceInKNB := PrgStation.stRecipeParams.stRecipeEnduranceRun.rLoadForceB;
  rTargetSpeedAInMmPerS := PrgStation.stRecipeParams.stRecipeEnduranceRun.rSpeedA;
  rTargetSpeedBInMmPerS := PrgStation.stRecipeParams.stRecipeEnduranceRun.rSpeedB;
  lrNokLimit := PrgStation.stRecipeParams.stRecipeEnduranceRun.stLT1_Params.rNokLimit;
ELSIF PrgVisu.fbVisuOPMode.P_BreakPressureDetSelected THEN
  sTagName := 'Losbrechdruck';
  liTargetCycles := PrgStation.stRecipeParams.stRecipeBreakPressure.uiVentCycles;
  rTargetTestPressureInBarA := 0.0;
  rTargetTestPressureInBarB := 0.0;
  rTargetTestForceInKNA := 0.0;
  rTargetTestForceInKNB := 0.0;
  rTargetCounterPressureInBarA := 0.0;
  rTargetCounterPressureInBarB := 0.0;
  rTargetCounterForceInKNA := 0.0;
  rTargetCounterForceInKNB := 0.0;
  rTargetSpeedAInMmPerS := PrgStation.stRecipeParams.stRecipeBreakPressure.rMinSpeedInMmPerS;
  rTargetSpeedBInMmPerS := PrgStation.stRecipeParams.stRecipeBreakPressure.rMinSpeedInMmPerS;
  lrNokLimit := PrgStation.stRecipeParams.stRecipeBreakPressure.rNokLimit;
ELSIF PrgVisu.fbVisuOPMode.P_LeakTest1Selected THEN
  sTagName := 'Dichtheitsprüfung1';
  liTargetCycles := PrgStation.stRecipeParams.stRecipeLeakTest1.uiVentCycles;
  rTargetTestPressureInBarA := 0.0;
  rTargetTestPressureInBarB := 0.0;
  rTargetTestForceInKNA := 0.0;
  rTargetTestForceInKNB := 0.0;
  rTargetCounterPressureInBarA := PrgStation.stRecipeParams.stRecipeLeakTest1.rLoadPressureA;
  rTargetCounterPressureInBarB := PrgStation.stRecipeParams.stRecipeLeakTest1.rLoadPressureB;
  rTargetCounterForceInKNA := PrgStation.stRecipeParams.stRecipeLeakTest1.rLoadForceA;
  rTargetCounterForceInKNB := PrgStation.stRecipeParams.stRecipeLeakTest1.rLoadForceB;
  rTargetSpeedAInMmPerS := 0.0;
  rTargetSpeedBInMmPerS := 0.0;
  lrNokLimit := PrgStation.stRecipeParams.stRecipeLeakTest1.rNokLimit;
ELSIF PrgVisu.fbVisuOPMode.P_LeakTest2Selected THEN
  sTagName := 'Dichtheitsprüfung2';
  liTargetCycles := PrgStation.stRecipeParams.stRecipeLeakTest2.uiVentCycles;
  rTargetTestPressureInBarA := PrgStation.stRecipeParams.stRecipeLeakTest2.rLoadPressureA;
  rTargetTestPressureInBarB := PrgStation.stRecipeParams.stRecipeLeakTest2.rLoadPressureB;
  rTargetTestForceInKNA := PrgStation.stRecipeParams.stRecipeLeakTest2.rLoadForceA;
  rTargetTestForceInKNB := PrgStation.stRecipeParams.stRecipeLeakTest2.rLoadForceB;
  rTargetCounterPressureInBarA := 0.0;
  rTargetCounterPressureInBarB := 0.0;
  rTargetCounterForceInKNA := 0.0;
  rTargetCounterForceInKNB := 0.0;
  rTargetSpeedAInMmPerS := 0.0;
  rTargetSpeedBInMmPerS := 0.0;
  lrNokLimit := PrgStation.stRecipeParams.stRecipeLeakTest2.rNokLimit;
END_IF

// Current Timestamp
sCurrentDateTime := CONCAT(TO_STRING(systemTime.wYear), '_');
sCurrentDateTime := CONCAT(sCurrentDateTime, TO_STRING(systemTime.wMonth));
sCurrentDateTime := CONCAT(sCurrentDateTime, '_');
sCurrentDateTime := CONCAT(sCurrentDateTime, TO_STRING(systemTime.wDay));
sCurrentDateTime := CONCAT(sCurrentDateTime, '_');
sCurrentDateTime := CONCAT(sCurrentDateTime, TO_STRING(systemTime.wHour));
sCurrentDateTime := CONCAT(sCurrentDateTime, '_');
sCurrentDateTime := CONCAT(sCurrentDateTime, TO_STRING(systemTime.wMinute));
sCurrentDateTime := CONCAT(sCurrentDateTime, '_');
sCurrentDateTime := CONCAT(sCurrentDateTime, TO_STRING(systemTime.wSecond));
END_ACTION

ACTION A_020_DBNest1:
// Assign Nest1 values to database
sMeasurementName := PrgStation.sTestCyl1SNo;

stFieldValues.sTimeStamp := sCurrentDateTime;
stFieldValues.sTimer := PrgStation.fbTimerNest1.M_GetTimerET(FALSE, '');
stFieldValues.liTargetCycles := liTargetCycles;
stFieldValues.liActiveCycle := PrgStation.fbMainProcess.P_CurrentCycleNest1;
stFieldValues.iTestDirection := PrgStation.fbTestCyl1.P_ActiveDirection;
stFieldValues.rTargetTestPressureInBarA := rTargetTestPressureInBarA;
stFieldValues.rTargetTestPressureInBarB := rTargetTestPressureInBarB;
stFieldValues.rCurrentTestPressureInBar := PrgStation.rPressureConverted_TestCyl1;
stFieldValues.rTargetTestForceInKNA := rTargetTestForceInKNA;
stFieldValues.rTargetTestForceInKNB := rTargetTestForceInKNB;
stFieldValues.rCurrentTestForceInKN := PrgStation.fbTestCyl1.P_CurrentForceInKN;
stFieldValues.rTestPressureAInBar := PrgStation.rPressureConverted_TestCyl1_A;
stFieldValues.rTestPressureBInBar := PrgStation.rPressureConverted_TestCyl1_B;
stFieldValues.rBreakawayPressureInBar := PrgStation.rPressureConverted_LowPressure;
stFieldValues.rBreakawayPressureAInBar := PrgStation.rPressureConverted_TestCyl1_BreakPressure_A;
stFieldValues.rBreakawayPressureBInBar := PrgStation.rPressureConverted_TestCyl1_BreakPressure_B;
stFieldValues.rReservoirPressureInBar := PrgStation.rPressureConverted_TestCyl1_PressureReservoir;
stFieldValues.rTargetCounterPressureInBarA := rTargetCounterPressureInBarA;
stFieldValues.rTargetCounterPressureInBarB := rTargetCounterPressureInBarB;
stFieldValues.rCurrentCounterPressureInBar := PrgStation.rPressureConverted_CounterCyl1;
stFieldValues.rTargetCounterForceInKNA := rTargetCounterForceInKNA;
stFieldValues.rTargetCounterForceInKNB := rTargetCounterForceInKNB;
stFieldValues.rCurrentCounterForceInKN := PrgStation.fbCounterCyl1.P_CurrentForceInKN;
stFieldValues.lrPosition := PrgStation.fbTestCyl1.P_Position;
stFieldValues.lrPositionMin := PrgStation.fbTestCyl1.P_MinPosVal;
stFieldValues.lrPositionMax := PrgStation.fbTestCyl1.P_MaxPosVal;
stFieldValues.lrCylStrokeLength := PrgStation.fbTestCyl1.P_StrokeLength;
stFieldValues.lrTemperature := 0; // Programmieren????
stFieldValues.lrCylPistonSurfaceA := PrgStation.stRecipeParams.stRecipeCyl.lrPistonSurfaceA;
stFieldValues.lrCylPistonSurfaceB := PrgStation.stRecipeParams.stRecipeCyl.lrPistonSurfaceB;
stFieldValues.lrNokLimit := lrNokLimit;
stFieldValues.lrCurrentNokDifference := PrgStation.fbNest1.P_NokDifference;
stFieldValues.lrCurrentNokLimitInPercent := PrgStation.fbNest1.P_NokLimitInPercent;
stFieldValues.lrTargetSpeedAInMmPerS := rTargetSpeedAInMmPerS;
stFieldValues.lrTargetSpeedBInMmPerS := rTargetSpeedBInMmPerS;
END_ACTION

ACTION A_030_DBNest2:
// Assign Nest2 values to database
sMeasurementName := PrgStation.sTestCyl2SNo;

stFieldValues.sTimeStamp := sCurrentDateTime;
stFieldValues.sTimer := PrgStation.fbTimerNest2.M_GetTimerET(FALSE, '');
stFieldValues.liTargetCycles := liTargetCycles;
stFieldValues.liActiveCycle := PrgStation.fbMainProcess.P_CurrentCycleNest2;
stFieldValues.iTestDirection := PrgStation.fbTestCyl2.P_ActiveDirection;
stFieldValues.rTargetTestPressureInBarA := rTargetTestPressureInBarA;
stFieldValues.rTargetTestPressureInBarB := rTargetTestPressureInBarB;
stFieldValues.rCurrentTestPressureInBar := PrgStation.rPressureConverted_TestCyl2;
stFieldValues.rTargetTestForceInKNA := rTargetTestForceInKNA;
stFieldValues.rTargetTestForceInKNB := rTargetTestForceInKNB;
stFieldValues.rCurrentTestForceInKN := PrgStation.fbTestCyl2.P_CurrentForceInKN;
stFieldValues.rTestPressureAInBar := PrgStation.rPressureConverted_TestCyl2_A;
stFieldValues.rTestPressureBInBar := PrgStation.rPressureConverted_TestCyl2_B;
stFieldValues.rBreakawayPressureInBar := 0.0;
stFieldValues.rBreakawayPressureAInBar := 0.0;
stFieldValues.rBreakawayPressureBInBar := 0.0;
stFieldValues.rReservoirPressureInBar := 0.0;
stFieldValues.rTargetCounterPressureInBarA := rTargetCounterPressureInBarA;
stFieldValues.rTargetCounterPressureInBarB := rTargetCounterPressureInBarB;
stFieldValues.rCurrentCounterPressureInBar := PrgStation.rPressureConverted_CounterCyl2;
stFieldValues.rTargetCounterForceInKNA := rTargetCounterForceInKNA;
stFieldValues.rTargetCounterForceInKNB := rTargetCounterForceInKNB;
stFieldValues.rCurrentCounterForceInKN := PrgStation.fbCounterCyl2.P_CurrentForceInKN;
stFieldValues.lrPosition := PrgStation.fbTestCyl2.P_Position;
stFieldValues.lrPositionMin := PrgStation.fbTestCyl2.P_MinPosVal;
stFieldValues.lrPositionMax := PrgStation.fbTestCyl2.P_MaxPosVal;
stFieldValues.lrCylStrokeLength := PrgStation.fbTestCyl2.P_StrokeLength;
stFieldValues.lrTemperature := 0; // Programmieren????
stFieldValues.lrCylPistonSurfaceA := PrgStation.stRecipeParams.stRecipeCyl.lrPistonSurfaceA;
stFieldValues.lrCylPistonSurfaceB := PrgStation.stRecipeParams.stRecipeCyl.lrPistonSurfaceB;
stFieldValues.lrNokLimit := lrNokLimit;
stFieldValues.lrCurrentNokDifference := PrgStation.fbNest2.P_NokDifference;
stFieldValues.lrCurrentNokLimitInPercent := PrgStation.fbNest2.P_NokLimitInPercent;
stFieldValues.lrTargetSpeedAInMmPerS := rTargetSpeedAInMmPerS;
stFieldValues.lrTargetSpeedBInMmPerS := rTargetSpeedBInMmPerS;
END_ACTION

ACTION A_040_DBNest3:
// Assign Nest3 values to database
sMeasurementName := PrgStation.sTestCyl3SNo;

stFieldValues.sTimeStamp := sCurrentDateTime;
stFieldValues.sTimer := PrgStation.fbTimerNest3.M_GetTimerET(FALSE, '');
stFieldValues.liTargetCycles := liTargetCycles;
stFieldValues.liActiveCycle := PrgStation.fbMainProcess.P_CurrentCycleNest3;
stFieldValues.iTestDirection := PrgStation.fbTestCyl3.P_ActiveDirection;
stFieldValues.rTargetTestPressureInBarA := rTargetTestPressureInBarA;
stFieldValues.rTargetTestPressureInBarB := rTargetTestPressureInBarB;
stFieldValues.rCurrentTestPressureInBar := PrgStation.rPressureConverted_TestCyl3;
stFieldValues.rTargetTestForceInKNA := rTargetTestForceInKNA;
stFieldValues.rTargetTestForceInKNB := rTargetTestForceInKNB;
stFieldValues.rCurrentTestForceInKN := PrgStation.fbTestCyl3.P_CurrentForceInKN;
stFieldValues.rTestPressureAInBar := PrgStation.rPressureConverted_TestCyl3_A;
stFieldValues.rTestPressureBInBar := PrgStation.rPressureConverted_TestCyl3_B;
stFieldValues.rBreakawayPressureInBar := 0.0;
stFieldValues.rBreakawayPressureAInBar := 0.0;
stFieldValues.rBreakawayPressureBInBar := 0.0;
stFieldValues.rReservoirPressureInBar := 0.0;
stFieldValues.rTargetCounterPressureInBarA := rTargetCounterPressureInBarA;
stFieldValues.rTargetCounterPressureInBarB := rTargetCounterPressureInBarB;
stFieldValues.rCurrentCounterPressureInBar := PrgStation.rPressureConverted_CounterCyl3;
stFieldValues.rTargetCounterForceInKNA := rTargetCounterForceInKNA;
stFieldValues.rTargetCounterForceInKNB := rTargetCounterForceInKNB;
stFieldValues.rCurrentCounterForceInKN := PrgStation.fbCounterCyl3.P_CurrentForceInKN;
stFieldValues.lrPosition := PrgStation.fbTestCyl3.P_Position;
stFieldValues.lrPositionMin := PrgStation.fbTestCyl3.P_MinPosVal;
stFieldValues.lrPositionMax := PrgStation.fbTestCyl3.P_MaxPosVal;
stFieldValues.lrCylStrokeLength := PrgStation.fbTestCyl3.P_StrokeLength;
stFieldValues.lrTemperature := 0; // Programmieren????
stFieldValues.lrCylPistonSurfaceA := PrgStation.stRecipeParams.stRecipeCyl.lrPistonSurfaceA;
stFieldValues.lrCylPistonSurfaceB := PrgStation.stRecipeParams.stRecipeCyl.lrPistonSurfaceB;
stFieldValues.lrNokLimit := lrNokLimit;
stFieldValues.lrCurrentNokDifference := PrgStation.fbNest3.P_NokDifference;
stFieldValues.lrCurrentNokLimitInPercent := PrgStation.fbNest3.P_NokLimitInPercent;
stFieldValues.lrTargetSpeedAInMmPerS := rTargetSpeedAInMmPerS;
stFieldValues.lrTargetSpeedBInMmPerS := rTargetSpeedBInMmPerS;
END_ACTION

ACTION A_050_DBNest4:
// Assign Nest3 values to database
sMeasurementName := PrgStation.sTestCyl4SNo;

stFieldValues.sTimeStamp := sCurrentDateTime;
stFieldValues.sTimer := PrgStation.fbTimerNest4.M_GetTimerET(FALSE, '');
stFieldValues.liTargetCycles := liTargetCycles;
stFieldValues.liActiveCycle := PrgStation.fbMainProcess.P_CurrentCycleNest4;
stFieldValues.iTestDirection := PrgStation.fbTestCyl4.P_ActiveDirection;
stFieldValues.rTargetTestPressureInBarA := rTargetTestPressureInBarA;
stFieldValues.rTargetTestPressureInBarB := rTargetTestPressureInBarB;
stFieldValues.rCurrentTestPressureInBar := PrgStation.rPressureConverted_TestCyl4;
stFieldValues.rTargetTestForceInKNA := rTargetTestForceInKNA;
stFieldValues.rTargetTestForceInKNB := rTargetTestForceInKNB;
stFieldValues.rCurrentTestForceInKN := PrgStation.fbTestCyl4.P_CurrentForceInKN;
stFieldValues.rTestPressureAInBar := PrgStation.rPressureConverted_TestCyl4_A;
stFieldValues.rTestPressureBInBar := PrgStation.rPressureConverted_TestCyl4_B;
stFieldValues.rBreakawayPressureInBar := 0.0;
stFieldValues.rBreakawayPressureAInBar := 0.0;
stFieldValues.rBreakawayPressureBInBar := 0.0;
stFieldValues.rReservoirPressureInBar := 0.0;
stFieldValues.rTargetCounterPressureInBarA := rTargetCounterPressureInBarA;
stFieldValues.rTargetCounterPressureInBarB := rTargetCounterPressureInBarB;
stFieldValues.rCurrentCounterPressureInBar := PrgStation.rPressureConverted_CounterCyl4;
stFieldValues.rTargetCounterForceInKNA := rTargetCounterForceInKNA;
stFieldValues.rTargetCounterForceInKNB := rTargetCounterForceInKNB;
stFieldValues.rCurrentCounterForceInKN := PrgStation.fbCounterCyl4.P_CurrentForceInKN;
stFieldValues.lrPosition := PrgStation.fbTestCyl4.P_Position;
stFieldValues.lrPositionMin := PrgStation.fbTestCyl4.P_MinPosVal;
stFieldValues.lrPositionMax := PrgStation.fbTestCyl4.P_MaxPosVal;
stFieldValues.lrCylStrokeLength := PrgStation.fbTestCyl4.P_StrokeLength;
stFieldValues.lrTemperature := 0; // Programmieren????
stFieldValues.lrCylPistonSurfaceA := PrgStation.stRecipeParams.stRecipeCyl.lrPistonSurfaceA;
stFieldValues.lrCylPistonSurfaceB := PrgStation.stRecipeParams.stRecipeCyl.lrPistonSurfaceB;
stFieldValues.lrNokLimit := lrNokLimit;
stFieldValues.lrCurrentNokDifference := PrgStation.fbNest4.P_NokDifference;
stFieldValues.lrCurrentNokLimitInPercent := PrgStation.fbNest4.P_NokLimitInPercent;
stFieldValues.lrTargetSpeedAInMmPerS := rTargetSpeedAInMmPerS;
stFieldValues.lrTargetSpeedBInMmPerS := rTargetSpeedBInMmPerS;
END_ACTION

ACTION A_100_SaveToDB:
(* Timer *)
// Abort condition
tonFailedSavelimitTimer(IN:= NOT tonFailedSavelimitTimer.Q, PT:= tFailedSaveLimitTime);
IF tonFailedSavelimitTimer.Q THEN
  uiFailedSaveCounter := 0;
ELSE
  IF uiFailedSaveCounter >= uiAllowedSaveFail THEN
    bRecord := FALSE;
    ;// Error and abort
	END_IF
END_IF

// Save to database
tonSwitchTimer();
tonInterval();
IF bRecord THEN
  // First xxmin save interval = 0.5s and then 2min
  tonSwitchTimer(IN:= TRUE, PT:= tSwitchTime);
  IF tonSwitchTimer.Q THEN
    uiAllowedSaveFail := 2;
    tInterval := T#2M;
  ELSE
    uiAllowedSaveFail := 10;
    tInterval := T#500MS;
  END_IF
  // Save interval
  tonInterval(IN:= TRUE, PT:= tInterval);
  IF tonInterval.Q AND NOT bSaveBusy THEN
    bSaveTrigger := TRUE;
  END_IF
ELSE
  // Reset
  tonSwitchTimer.IN := FALSE;
  tonInterval.IN := FALSE;
  //iSaveSeq := 0;
END_IF
// Save action
IF bSaveTrigger THEN
  bSaveBusy := TRUE;
  CASE iSaveSeq OF
    0:
      IF fbInfluxDB.M_SetReady() THEN
          iSeqCounter := iSeqCounter + 1;
          iSaveSeq := iSeqCounter;
      END_IF
    1:
      A_020_DBNest1();
      IF PrgStation.fbNest1.bEnable THEN
        IF TRUE
        AND fbInfluxDB.M_WriteStruct(sBucketName:= sBucketName,
                                    sMeasurementName:= sMeasurementName,
                                    sTagName:= sTagName,
                                    stFieldValues:= stFieldValues,
                                    bResult=> bSaveSuccess) 
        THEN
          IF bSaveSuccess THEN
            bSaveSuccess := FALSE;
          ELSE
            // Warningmessage/-log, but no abort (Abort with tonFailedSavelimitTimer)
            // ...
            uiFailedSaveCounter := uiFailedSaveCounter + 1;
					END_IF
          iSaveSeq := 0;
        END_IF
      ELSE
        iSaveSeq := 0;
      END_IF
    2:
      A_030_DBNest2();
      IF PrgStation.fbNest2.bEnable THEN
        IF TRUE
        AND fbInfluxDB.M_WriteStruct(sBucketName:= sBucketName,
                                    sMeasurementName:= sMeasurementName,
                                    sTagName:= sTagName,
                                    stFieldValues:= stFieldValues,
                                    bResult=> bSaveSuccess) 
        THEN
          IF bSaveSuccess THEN
            bSaveSuccess := FALSE;
          ELSE
            // Warningmessage/-log, but no abort (Abort with tonFailedSavelimitTimer)
            // ...
            uiFailedSaveCounter := uiFailedSaveCounter + 1;
					END_IF
          iSaveSeq := 0;
        END_IF
      ELSE
        iSaveSeq := 0;
      END_IF
    3:
      A_040_DBNest3();
      IF PrgStation.fbNest3.bEnable THEN
        IF TRUE
        AND fbInfluxDB.M_WriteStruct(sBucketName:= sBucketName,
                                    sMeasurementName:= sMeasurementName,
                                    sTagName:= sTagName,
                                    stFieldValues:= stFieldValues,
                                    bResult=> bSaveSuccess) 
        THEN
          IF bSaveSuccess THEN
            bSaveSuccess := FALSE;
          ELSE
            // Warningmessage/-log, but no abort (Abort with tonFailedSavelimitTimer)
            // ...
            uiFailedSaveCounter := uiFailedSaveCounter + 1;
					END_IF
          iSaveSeq := 0;
        END_IF
      ELSE
        iSaveSeq := 0;
      END_IF
    4:
      A_050_DBNest4();
      IF PrgStation.fbNest4.bEnable THEN
        IF TRUE
        AND fbInfluxDB.M_WriteStruct(sBucketName:= sBucketName,
                                    sMeasurementName:= sMeasurementName,
                                    sTagName:= sTagName,
                                    stFieldValues:= stFieldValues,
                                    bResult=> bSaveSuccess) 
        THEN
          IF bSaveSuccess THEN
            bSaveSuccess := FALSE;
          ELSE
            // Warningmessage/-log, but no abort (Abort with tonFailedSavelimitTimer)
            // ...
            uiFailedSaveCounter := uiFailedSaveCounter + 1;
					END_IF
          iSaveSeq := 0;
        END_IF
      END_IF
      iSaveSeq := 0;
      iSeqCounter := 0;
      bSaveTrigger := FALSE;
      tonInterval.IN := FALSE;
      bSaveBusy := FALSE;
  END_CASE
END_IF
END_ACTION

ACTION A_110_TotalMeasurements:
IF bGetTotalMeasurements THEN
  CASE uiTotalMeasurementsSeq OF
    0:
      IF fbInfluxDB.M_SetReady() THEN
          uiTotalMeasurementsSeq := 1;
      END_IF
    1:
      IF fbInfluxDB.M_GetTotalMeasurements(sBucketName:= sBucketName, 
                                           bResult=> bGetTotalMeasurementsProcessSuccess, 
                                           uiResult=> uiTotalMeasurements) 
      THEN
        IF bGetTotalMeasurementsProcessSuccess THEN
          bGetTotalMeasurementsProcessSuccess := FALSE;
        ELSE
          // Warningmessage/-log, but no abort (Abort with tonFailedSavelimitTimer)
          // ...
				END_IF
        bGetTotalMeasurements := FALSE;
        uiTotalMeasurementsSeq := 0;
			END_IF
	END_CASE
END_IF
END_ACTION

ACTION A_120_MeasurementExistCheck:
// Init

// General
IF bGetMeasurementExist THEN
  CASE uiMeasurementExistSeq OF
    0:
      IF fbInfluxDB.M_SetReady() THEN
          uiMeasurementExistSeq := 1;
      END_IF
    1:
      IF fbInfluxDB.M_MeasurementExistCheck(sBucketName:= sBucketName,
                                            sMeasurementName:= sMeasurementNameFromCfg, 
                                            bResult=> bMeasurementExist) 
      THEN
        bGetMeasurementExist := FALSE;
        uiMeasurementExistSeq := 0;
			END_IF
	END_CASE
END_IF
END_ACTION

ACTION A_130_TagExistCheck:
// Init
CASE uiTagNameIDFromCfg OF
  1:
    sTagNameFromCfg := 'Dauerlauf';
  2:
    sTagNameFromCfg := 'Dichtheitsprüfung1';
  3:
    sTagNameFromCfg := 'Dichtheitsprüfung2';
  4:
    sTagNameFromCfg := 'Losbrechdruck';
  5:
    sTagNameFromCfg := '';
END_CASE

// General
IF bGetTagExist THEN
  CASE uiTagExistSeq OF
    0:
      IF fbInfluxDB.M_SetReady() THEN
          uiTagExistSeq := 1;
      END_IF
    1:
      IF fbInfluxDB.M_TagExistCheck(sBucketName:= sBucketName,
                                    sMeasurementName:= sMeasurementNameFromCfg,
                                    sTagName:= sTagNameFromCfg, 
                                    bResult=> bTagExist) 
      THEN
        bGetTagExist := FALSE;
        uiTagExistSeq := 0;
			END_IF
	END_CASE
END_IF
END_ACTION

ACTION A_140_DeleteMeasurement:
// Init

// General
IF bDeleteMeasurement THEN
  CASE uiDeleteMeasurementSeq OF
    0:
      IF fbInfluxDB.M_SetReady() THEN
        uiDeleteMeasurementSeq := 1;
      END_IF
    1:
      IF fbInfluxDB.M_DeleteMeasurement(sBucketName:= sBucketName,
                                        sMeasurementName:= sMeasurementNameFromCfg, 
                                        bResult=> bDeleteMeasurementResult) 
      THEN
        bDeleteMeasurement := FALSE;
        uiDeleteMeasurementSeq := 0;
			END_IF
	END_CASE
END_IF
END_ACTION

ACTION A_150_DeleteTag:
// Init
CASE uiTagNameIDFromCfg OF
  1:
    sTagNameFromCfg := 'Dauerlauf';
  2:
    sTagNameFromCfg := 'Dichtheitsprüfung1';
  3:
    sTagNameFromCfg := 'Dichtheitsprüfung2';
  4:
    sTagNameFromCfg := 'Losbrechdruck';
  5:
    sTagNameFromCfg := '';
END_CASE

// General
IF bDeleteTag THEN
  CASE uiDeleteTagSeq OF
    0:
      IF fbInfluxDB.M_SetReady() THEN
        uiDeleteTagSeq := 1;
      END_IF
    1:
      IF fbInfluxDB.M_DeleteTag(sBucketName:= sBucketName,
                                        sMeasurementName:= sMeasurementNameFromCfg, 
                                        sTagName:= sTagNameFromCfg,
                                        bResult=> bDeleteTagResult) 
      THEN
        bDeleteTag := FALSE;
        uiDeleteTagSeq := 0;
			END_IF
	END_CASE
END_IF
END_ACTION

ACTION A_160_DeleteTagContentBlock:
// Init
CASE uiTagNameIDFromCfg OF
  1:
    sTagNameFromCfg := 'Dauerlauf';
  2:
    sTagNameFromCfg := 'Dichtheitsprüfung1';
  3:
    sTagNameFromCfg := 'Dichtheitsprüfung2';
  4:
    sTagNameFromCfg := 'Losbrechdruck';
  5:
    sTagNameFromCfg := '';
END_CASE

// General
IF bDeleteTagContentBlock THEN
  CASE uiDeleteTagContentBlockSeq OF
    0:
      IF fbInfluxDB.M_SetReady() THEN
        uiDeleteTagContentBlockSeq := 1;
      END_IF
    1:
      IF fbInfluxDB.M_DeleteTagContentBlock(sBucketName:= sBucketName,
                                            sMeasurementName:= sMeasurementNameFromCfg, 
                                            sTagName:= sTagNameFromCfg,
                                            dtFrom:= dtFromFromCfg,
                                            dtTo:= dtToFromCfg,
                                            bResult=> bDeleteTagContentBlockResult) 
      THEN
        bDeleteTagContentBlock := FALSE;
        uiDeleteTagContentBlockSeq := 0;
			END_IF
	END_CASE
END_IF
END_ACTION

END_PROGRAM

// ---- MODULE/DATABASE/POU/FB_INFLUX_DB_ADS.TcPOU
FUNCTION_BLOCK FB_INFLUX_DB_ADS IMPLEMENTS I_INFLUXDB_ADS
VAR_IN_OUT
  bResult:                                                BOOL;
END_VAR
VAR_INPUT
  bADSLifeBit:                                            BOOL;
  bAdsConnected:                                          BOOL;
  bReady:                                                 BOOL;
  bBusy:                                                  BOOL;
END_VAR
VAR //General
	{attribute 'instance-path'} 
  {attribute 'noinit'} 
	strInstancePath:									                      STRING;
	bInit: 												                          BOOL:=TRUE;
	strFullObjectPath: 								                      STRING;
	stEvent:											                          ST_EVENT;
	bAck:												                            BOOL;
	
END_VAR
VAR   // From FB_init	
	itfOpMode:											                        I_OP_MODE; 
  itfEventLogger:                                         I_EVENT_LOGGER;
END_VAR                                      				
VAR	// Step chain control                				
  eSeq, eLastSeq, eNextSeq:					                      E_SEQ_DATABASE; 
  i:														                          INT;
  stSeqCtrlGeneral:											                  ST_SEQ_CTRL_GEN;     	
END_VAR                                             		
VAR                                                 		
	bMethodeFromExtStarted:									                BOOL;
	bMethodeFromExtActive:									                BOOL;
	bMethodeFromExtDone:									                  BOOL;
	strTemp:												                        STRING;
END_VAR   
VAR
  // From ADS
  bDBLifeBit:                                             BOOL;
  liDatabaseSizeInMb:                                     LINT;
  udiDatabaseSizeInMb:                                    UDINT;
  uiTotalMeasurements:                                    UINT;
  // To ADS
  bGetBucketExist:                                        BOOL;
  sBucketName:                                            T_MaxString := '3925-HZP';
  bGetMeasurementExist:                                   BOOL;
  sMeasurementName:                                       T_MaxString;
  bDeleteMeasurement:                                     BOOL;
  bDeleteAllMeasurements:                                 BOOL;
  bWriteStructData:                                       BOOL;
  sTagName:                                               T_MaxString;
  sFieldName:                                             T_MaxString;
  stFieldValues:                                          ST_DATABASE_RECORD;
  pFieldStructContent:                                    POINTER TO ARRAY [0..99] OF T_MaxString;
  pFieldNames:                                            POINTER TO ARRAY [0..99] OF T_MaxString;
  dtFrom:                                                 DT;
  dtTo:                                                   DT;
  sDtFrom:                                                T_MaxString;
  sDtTo:                                                  T_MaxString;
  sFieldNameExistCheck:                                   T_MaxString;
  bGetTagExist:                                           BOOL;
  bGetFieldExist:                                         BOOL;
  bClearMeasurement:                                      BOOL;
  bDeleteTag:                                             BOOL;
  bDeleteTagContentBlock:                                 BOOL;
  bDeleteField:                                           BOOL;
  bGetTotalMeasurements:                                  BOOL;
END_VAR    
VAR // State
  tLifeBitTimeout:                                        TIME := T#5S;
  // ADS
  uiADSStateSeq:                                          UINT := 0;
  tonADSState:                                            TON;
  bResetADSStateTimer:                                    BOOL;
  bADSState:                                              BOOL := TRUE;
  // InfluxDB
  uiInfluxDBStateSeq:                                     UINT := 0;
  tonInfluxDBState:                                       TON;
  bResetInfluxDBStateTimer:                               BOOL;
  bInfluxDBState:                                         BOOL := TRUE;
END_VAR              	
VAR_TEMP                    	
	iTemp:										                              INT;
END_VAR

// Set FBs and Interfaces ready after switch internal step
IF stSeqCtrlGeneral.iInternalSeqStateCase <> stSeqCtrlGeneral.iLastInternalSeqStateCase AND NOT stSeqCtrlGeneral.bExitSetReadyState THEN
  IF TRUE
  THEN
    stSeqCtrlGeneral.bExitSetReadyState := TRUE;
  ELSE
    RETURN;
  END_IF
END_IF

stSeqCtrlGeneral.strObject := F_CreateObjectName(strInstancePath);

// Init
// Format Time string for InfluxDB
sDtFrom := DT_TO_STRING(dtFrom);
sDtFrom := DELETE(sDtFrom, 3, 1);
sDtFrom := REPLACE(sDtFrom, 'T', 1, 11);
sDtFrom := CONCAT(sDtFrom, 'Z');
sDtTo := DT_TO_STRING(dtTo);
sDtTo := DELETE(sDtTo, 3, 1);
sDtTo := REPLACE(sDtTo, 'T', 1, 11);
sDtTo := CONCAT(sDtTo, 'Z');

// Actions
A_010_ADSState();
A_020_InfluxDBState();

// First method call
_m_SequenceManager();
//_m_SaveLastStep();

udiDatabaseSizeInMb := TO_UDINT(liDatabaseSizeInMb);

CASE eSeq OF 
  E_SEQ_DATABASE.BASE:;
  
	E_SEQ_DATABASE.INIT: _m_Seq_INIT();
		IF TRUE
		AND (stSeqCtrlGeneral.eActiveSeqState = E_SEQ_GENERAL.DONE) 
		THEN
			eSeq := E_SEQ_DATABASE.BASE;
		END_IF
		
	E_SEQ_DATABASE.SETUP:;
  
